C01778=1020.388,138.812,-115.444,167.637,51.113,159.489
C01779=1020.383,138.562,-115.424,167.634,51.119,159.489
C01780=1020.377,138.313,-115.404,167.630,51.126,159.490
C01781=1020.372,138.063,-115.384,167.627,51.133,159.491
C01782=1020.366,137.814,-115.364,167.624,51.140,159.492
C01783=1020.361,137.565,-115.344,167.621,51.147,159.493
C01784=1020.356,137.316,-115.324,167.618,51.154,159.493
C01785=1020.350,137.067,-115.305,167.614,51.160,159.494
C01786=1020.345,136.818,-115.285,167.611,51.167,159.495
C01787=1020.339,136.568,-115.265,167.609,51.174,159.496
C01788=1020.334,136.319,-115.245,167.605,51.181,159.497
C01789=1020.329,136.070,-115.226,167.602,51.188,159.497
C01790=1020.324,135.821,-115.205,167.599,51.195,159.498
C01791=1020.318,135.572,-115.186,167.596,51.201,159.499
C01792=1020.313,135.323,-115.165,167.593,51.208,159.500
C01793=1020.308,135.074,-115.147,167.590,51.215,159.501
C01794=1020.303,134.824,-115.127,167.586,51.222,159.501
C01795=1020.297,134.575,-115.107,167.583,51.229,159.502
C01796=1020.292,134.326,-115.087,167.581,51.236,159.503
C01797=1020.287,134.078,-115.067,167.578,51.243,159.504
C01798=1020.282,133.828,-115.048,167.574,51.250,159.505
C01799=1020.276,133.578,-115.028,167.571,51.257,159.505
C01800=1020.270,133.330,-115.008,167.569,51.263,159.506
C01801=1020.266,133.081,-114.989,167.565,51.270,159.507
C01802=1020.260,132.831,-114.970,167.562,51.277,159.508
C01803=1020.255,132.582,-114.949,167.559,51.284,159.509
C01804=1020.249,132.333,-114.930,167.556,51.290,159.510
C01805=1020.245,132.084,-114.910,167.553,51.297,159.510
C01806=1020.239,131.835,-114.890,167.550,51.304,159.511
C01807=1020.234,131.585,-114.871,167.546,51.311,159.512
C01808=1020.229,131.336,-114.852,167.544,51.318,159.513
C01809=1020.223,131.087,-114.832,167.541,51.325,159.514
C01810=1020.218,130.838,-114.812,167.537,51.331,159.514
C01811=1020.212,130.588,-114.793,167.534,51.338,159.515
C01812=1020.208,130.339,-114.773,167.532,51.345,159.516
C01813=1020.202,130.090,-114.754,167.528,51.352,159.517
C01814=1020.197,129.841,-114.733,167.525,51.359,159.518
C01815=1020.191,129.591,-114.714,167.522,51.366,159.518
C01816=1020.186,129.343,-114.695,167.520,51.373,159.519
C01817=1020.180,129.093,-114.676,167.516,51.380,159.520
C01818=1020.175,128.844,-114.657,167.513,51.387,159.521
C01819=1020.169,128.595,-114.638,167.510,51.394,159.522
C01820=1020.164,128.346,-114.619,167.506,51.401,159.522
C01821=1020.158,128.096,-114.599,167.504,51.407,159.523
C01822=1020.153,127.847,-114.581,167.501,51.415,159.524
C01823=1020.148,127.598,-114.561,167.498,51.422,159.525
C01824=1020.142,127.348,-114.541,167.495,51.429,159.526
C01825=1020.137,127.099,-114.523,167.491,51.436,159.527
C01826=1020.132,126.850,-114.503,167.489,51.442,159.528
C01827=1020.126,126.601,-114.484,167.486,51.450,159.529
C01828=1020.121,126.352,-114.465,167.483,51.457,159.529
C01829=1020.115,126.102,-114.446,167.479,51.464,159.530
C01830=1020.109,125.853,-114.427,167.477,51.470,159.531
C01831=1020.104,125.604,-114.408,167.474,51.477,159.532
C01832=1020.099,125.355,-114.389,167.470,51.484,159.533
C01833=1020.094,125.106,-114.370,167.467,51.491,159.533
C01834=1020.089,124.856,-114.350,167.465,51.498,159.534
C01835=1020.083,124.607,-114.331,167.462,51.505,159.535
C01836=1020.078,124.358,-114.312,167.459,51.512,159.536
C01837=1020.072,124.109,-114.293,167.455,51.519,159.537
C01838=1020.067,123.860,-114.274,167.453,51.526,159.538
C01839=1020.061,123.577,-114.252,167.449,51.534,159.538
C01840=1020.054,123.294,-114.230,167.446,51.541,159.539
C01841=1020.048,123.011,-114.208,167.442,51.549,159.540
C01842=1020.042,122.729,-114.187,167.439,51.557,159.541
C01843=1020.037,122.480,-114.168,167.436,51.564,159.542
C01844=1020.032,122.230,-114.148,167.433,51.571,159.543
C01845=1020.027,121.982,-114.129,167.430,51.578,159.544
C01846=1020.021,121.732,-114.110,167.428,51.585,159.545
C01847=1020.016,121.484,-114.091,167.424,51.592,159.545
C01848=1020.010,121.234,-114.072,167.421,51.599,159.546
C01849=1020.005,120.985,-114.054,167.419,51.606,159.547
C01850=1020.000,120.735,-114.035,167.416,51.612,159.548
C01851=1019.994,120.486,-114.015,167.412,51.619,159.549
C01852=1019.989,120.237,-113.997,167.410,51.626,159.550
C01853=1019.983,119.988,-113.977,167.407,51.633,159.550
C01854=1019.978,119.739,-113.958,167.403,51.640,159.551
C01855=1019.972,119.490,-113.939,167.401,51.647,159.552
C01856=1019.968,119.240,-113.920,167.398,51.654,159.553
C01857=1019.963,118.990,-113.901,167.395,51.660,159.554
C01858=1019.958,118.742,-113.882,167.392,51.667,159.554
C01859=1019.952,118.492,-113.863,167.389,51.675,159.555
C01860=1019.947,118.244,-113.844,167.386,51.682,159.556
C01861=1019.941,117.993,-113.826,167.384,51.688,159.557
C01862=1019.936,117.745,-113.807,167.381,51.695,159.558
C01863=1019.931,117.495,-113.788,167.377,51.702,159.559
C01864=1019.926,117.247,-113.769,167.375,51.709,159.560
C01865=1019.920,116.997,-113.749,167.372,51.716,159.560
C01866=1019.915,116.748,-113.731,167.369,51.723,159.561
C01867=1019.909,116.498,-113.712,167.366,51.729,159.562
C01868=1019.904,116.250,-113.693,167.363,51.736,159.563
C01869=1019.899,116.001,-113.674,167.361,51.743,159.564
C01870=1019.894,115.751,-113.656,167.358,51.750,159.564
C01871=1019.890,115.502,-113.636,167.354,51.757,159.565
C01872=1019.884,115.252,-113.617,167.352,51.764,159.566
C01873=1019.879,115.004,-113.598,167.349,51.771,159.567
C01874=1019.873,114.754,-113.580,167.345,51.778,159.568
C01875=1019.868,114.505,-113.561,167.343,51.784,159.568
C01876=1019.863,114.255,-113.541,167.340,51.791,159.569
C01877=1019.858,114.006,-113.523,167.338,51.798,159.570
C01878=1019.853,113.757,-113.504,167.334,51.804,159.571
C01879=1019.847,113.508,-113.485,167.332,51.811,159.572
C01880=1019.842,113.259,-113.467,167.329,51.818,159.572
C01881=1019.837,113.009,-113.448,167.325,51.825,159.573
C01882=1019.832,112.760,-113.429,167.323,51.831,159.574
C01883=1019.827,112.511,-113.411,167.320,51.838,159.575
C01884=1019.821,112.262,-113.391,167.318,51.845,159.576
C01885=1019.816,112.012,-113.373,167.314,51.852,159.576
C01886=1019.811,111.763,-113.354,167.311,51.859,159.577
C01887=1019.806,111.513,-113.336,167.309,51.866,159.578
C01888=1019.799,111.264,-113.317,167.306,51.873,159.579
C01889=1019.795,111.015,-113.299,167.303,51.880,159.580
C01890=1019.790,110.766,-113.280,167.301,51.887,159.581
C01891=1019.784,110.516,-113.262,167.297,51.894,159.582
C01892=1019.778,110.268,-113.243,167.294,51.901,159.582
C01893=1019.774,110.018,-113.225,167.292,51.908,159.583
C01894=1019.768,109.769,-113.206,167.289,51.915,159.584
C01895=1019.763,109.520,-113.188,167.286,51.921,159.585
C01896=1019.757,109.271,-113.169,167.283,51.928,159.586
C01897=1019.752,109.021,-113.151,167.280,51.935,159.586
C01898=1019.747,108.772,-113.133,167.277,51.943,159.587
C01899=1019.741,108.523,-113.114,167.275,51.950,159.588
C01900=1019.736,108.273,-113.096,167.272,51.957,159.589
C01901=1019.730,108.024,-113.078,167.268,51.964,159.590
C01902=1019.725,107.775,-113.059,167.266,51.970,159.591
C01903=1019.719,107.492,-113.039,167.262,51.978,159.592
C01904=1019.712,107.209,-113.018,167.260,51.986,159.593
C01905=1019.706,106.927,-112.997,167.257,51.994,159.594
C01906=1019.700,106.644,-112.977,167.253,52.002,159.594
C01907=1019.695,106.395,-112.959,167.250,52.009,159.595
C01908=1019.689,106.146,-112.940,167.248,52.016,159.596
C01909=1019.684,105.896,-112.922,167.245,52.023,159.597
C01910=1019.679,105.647,-112.904,167.242,52.030,159.598
C01911=1019.674,105.398,-112.886,167.239,52.037,159.599
C01912=1019.668,105.148,-112.867,167.236,52.044,159.599
C01913=1019.663,104.899,-112.849,167.234,52.050,159.600
C01914=1019.658,104.650,-112.831,167.231,52.057,159.601
C01915=1019.652,104.400,-112.813,167.227,52.064,159.602
C01916=1019.647,104.151,-112.794,167.225,52.071,159.603
C01917=1019.641,103.902,-112.777,167.222,52.078,159.604
C01918=1019.636,103.652,-112.758,167.220,52.085,159.604
C01919=1019.631,103.403,-112.740,167.217,52.093,159.605
C01920=1019.625,103.155,-112.722,167.214,52.100,159.606
C01921=1019.620,102.905,-112.704,167.211,52.106,159.607
C01922=1019.614,102.655,-112.686,167.208,52.113,159.608
C01923=1019.609,102.406,-112.667,167.206,52.120,159.609
C01924=1019.604,102.157,-112.650,167.203,52.127,159.610
C01925=1019.599,101.908,-112.631,167.200,52.134,159.610
C01926=1019.593,101.658,-112.612,167.197,52.141,159.611
C01927=1019.588,101.409,-112.595,167.194,52.148,159.612
C01928=1019.583,101.160,-112.577,167.192,52.154,159.613
C01929=1019.578,100.911,-112.559,167.189,52.161,159.614
C01930=1019.572,100.661,-112.541,167.187,52.168,159.615
C01931=1019.566,100.412,-112.522,167.183,52.175,159.615
C01932=1019.562,100.163,-112.504,167.180,52.182,159.616
C01933=1019.557,99.914,-112.486,167.178,52.189,159.617
C01934=1019.551,99.664,-112.468,167.175,52.196,159.618
C01935=1019.546,99.415,-112.450,167.173,52.203,159.619
C01936=1019.540,99.166,-112.432,167.170,52.210,159.619
C01937=1019.536,98.916,-112.414,167.166,52.217,159.620
C01938=1019.529,98.666,-112.396,167.164,52.223,159.621
C01939=1019.524,98.417,-112.379,167.161,52.230,159.622
C01940=1019.518,98.168,-112.361,167.159,52.237,159.623
C01941=1019.514,97.919,-112.343,167.156,52.245,159.624
C01942=1019.508,97.670,-112.325,167.153,52.252,159.625
C01943=1019.502,97.420,-112.307,167.151,52.259,159.625
C01944=1019.496,97.171,-112.290,167.147,52.266,159.626
C01945=1019.492,96.922,-112.272,167.144,52.273,159.627
C01946=1019.486,96.673,-112.254,167.142,52.279,159.628
C01947=1019.481,96.424,-112.237,167.139,52.286,159.629
C01948=1019.476,96.173,-112.219,167.136,52.293,159.629
C01949=1019.470,95.924,-112.201,167.134,52.301,159.630
C01950=1019.465,95.675,-112.184,167.131,52.308,159.631
C01951=1019.459,95.426,-112.166,167.129,52.315,159.632
C01952=1019.454,95.177,-112.148,167.126,52.322,159.633
C01953=1019.448,94.927,-112.130,167.122,52.329,159.634
C01954=1019.443,94.678,-112.112,167.120,52.335,159.635
C01955=1019.437,94.429,-112.095,167.117,52.343,159.635
C01956=1019.432,94.179,-112.077,167.115,52.349,159.636
C01957=1019.427,93.930,-112.060,167.112,52.356,159.637
C01958=1019.422,93.681,-112.042,167.108,52.363,159.638
C01959=1019.417,93.431,-112.024,167.106,52.370,159.639
C01960=1019.411,93.182,-112.006,167.103,52.377,159.639
C01961=1019.405,92.933,-111.989,167.101,52.384,159.640
C01962=1019.400,92.684,-111.971,167.098,52.391,159.641
C01963=1019.395,92.434,-111.953,167.096,52.398,159.642
C01964=1019.390,92.185,-111.936,167.093,52.405,159.643
C01965=1019.384,91.936,-111.918,167.090,52.412,159.644
C01966=1019.379,91.687,-111.901,167.088,52.419,159.645
C01967=1019.373,91.404,-111.881,167.084,52.426,159.645
C01968=1019.367,91.121,-111.860,167.081,52.434,159.646
C01969=1019.361,90.839,-111.841,167.078,52.442,159.647
C01970=1019.354,90.555,-111.821,167.075,52.450,159.648
C01971=1019.349,90.306,-111.803,167.072,52.457,159.649
C01972=1019.343,90.057,-111.786,167.070,52.464,159.650
C01973=1019.339,89.808,-111.767,167.067,52.471,159.651
C01974=1019.333,89.558,-111.751,167.064,52.478,159.652
C01975=1019.328,89.309,-111.733,167.062,52.485,159.652
C01976=1019.323,89.060,-111.715,167.058,52.492,159.653
C01977=1019.317,88.811,-111.699,167.056,52.498,159.654
C01978=1019.312,88.561,-111.681,167.054,52.506,159.655
C01979=1019.306,88.312,-111.663,167.050,52.513,159.656
C01980=1019.301,88.063,-111.647,167.048,52.520,159.657
C01981=1019.295,87.813,-111.629,167.045,52.527,159.658
C01982=1019.290,87.563,-111.612,167.043,52.534,159.658
C01983=1019.284,87.314,-111.594,167.040,52.541,159.659
C01984=1019.279,87.065,-111.577,167.037,52.548,159.660
C01985=1019.273,86.816,-111.560,167.035,52.555,159.661
C01986=1019.268,86.567,-111.542,167.032,52.563,159.662
C01987=1019.263,86.317,-111.525,167.029,52.570,159.663
C01988=1019.257,86.068,-111.508,167.027,52.576,159.664
C01989=1019.252,85.818,-111.491,167.023,52.583,159.664
C01990=1019.246,85.569,-111.473,167.021,52.590,159.665
C01991=1019.241,85.320,-111.457,167.018,52.597,159.666
C01992=1019.236,85.070,-111.439,167.015,52.604,159.667
C01993=1019.230,84.821,-111.422,167.013,52.611,159.668
C01994=1019.225,84.572,-111.405,167.010,52.618,159.668
C01995=1019.220,84.322,-111.388,167.008,52.625,159.669
C01996=1019.214,84.073,-111.370,167.005,52.633,159.670
C01997=1019.208,83.824,-111.354,167.002,52.640,159.671
C01998=1019.203,83.575,-111.336,167.000,52.647,159.672
C01999=1019.197,83.325,-111.320,166.997,52.654,159.673
C02000=1019.192,83.076,-111.302,166.995,52.661,159.674
C02001=1019.187,82.826,-111.285,166.991,52.668,159.674
C02002=1019.181,82.577,-111.268,166.989,52.674,159.675
C02003=1019.176,82.328,-111.251,166.986,52.681,159.676
C02004=1019.171,82.078,-111.234,166.983,52.689,159.677
C02005=1019.165,81.829,-111.216,166.981,52.695,159.678
C02006=1019.160,81.579,-111.199,166.978,52.702,159.679
C02007=1019.155,81.330,-111.182,166.976,52.709,159.679
C02008=1019.149,81.081,-111.165,166.973,52.716,159.680
C02009=1019.144,80.832,-111.147,166.971,52.723,159.681
C02010=1019.139,80.582,-111.131,166.967,52.730,159.682
C02011=1019.133,80.332,-111.114,166.964,52.737,159.683
C02012=1019.128,80.083,-111.096,166.962,52.744,159.684
C02013=1019.123,79.834,-111.079,166.959,52.751,159.684
C02014=1019.116,79.585,-111.062,166.957,52.758,159.685
C02015=1019.111,79.335,-111.045,166.954,52.765,159.686
C02016=1019.106,79.085,-111.029,166.952,52.772,159.687
C02017=1019.100,78.836,-111.011,166.949,52.779,159.688
C02018=1019.095,78.587,-110.994,166.947,52.786,159.689
C02019=1019.091,78.338,-110.978,166.943,52.793,159.689
C02020=1019.085,78.089,-110.960,166.941,52.800,159.690
C02021=1019.080,77.839,-110.943,166.938,52.807,159.691
C02022=1019.075,77.589,-110.926,166.936,52.813,159.692
C02023=1019.069,77.340,-110.909,166.933,52.821,159.693
C02024=1019.064,77.091,-110.892,166.931,52.827,159.694
C02025=1019.058,76.841,-110.876,166.928,52.835,159.694
C02026=1019.052,76.592,-110.858,166.925,52.842,159.695
C02027=1019.047,76.343,-110.841,166.923,52.848,159.696
C02028=1019.042,76.093,-110.825,166.920,52.856,159.697
C02029=1019.036,75.844,-110.808,166.918,52.862,159.698
C02030=1019.031,75.594,-110.791,166.914,52.869,159.699
C02031=1019.025,75.313,-110.772,166.912,52.877,159.700
C02032=1019.019,75.030,-110.753,166.908,52.886,159.700
C02033=1019.013,74.747,-110.734,166.906,52.893,159.701
C02034=1019.007,74.465,-110.716,166.903,52.901,159.702
C02035=1019.001,74.215,-110.699,166.900,52.908,159.703
C02036=1018.996,73.966,-110.682,166.897,52.916,159.704
C02037=1018.991,73.716,-110.666,166.895,52.922,159.705
C02038=1018.984,73.467,-110.649,166.892,52.929,159.706
C02039=1018.979,73.218,-110.632,166.889,52.936,159.706
C02040=1018.974,72.968,-110.615,166.886,52.943,159.707
C02041=1018.969,72.719,-110.599,166.884,52.950,159.708
C02042=1018.963,72.470,-110.582,166.881,52.957,159.709
C02043=1018.957,72.220,-110.566,166.878,52.964,159.710
C02044=1018.952,71.971,-110.549,166.876,52.971,159.711
C02045=1018.947,71.721,-110.532,166.873,52.978,159.711
C02046=1018.941,71.472,-110.516,166.871,52.985,159.712
C02047=1018.936,71.223,-110.499,166.868,52.992,159.713
C02048=1018.931,70.973,-110.483,166.866,52.999,159.714
C02049=1018.925,70.724,-110.466,166.863,53.006,159.715
C02050=1018.920,70.474,-110.449,166.860,53.013,159.716
C02051=1018.914,70.225,-110.433,166.858,53.020,159.716
C02052=1018.909,69.975,-110.416,166.855,53.027,159.717
C02053=1018.904,69.726,-110.400,166.853,53.034,159.718
C02054=1018.898,69.477,-110.384,166.849,53.041,159.719
C02055=1018.893,69.227,-110.367,166.847,53.048,159.720
C02056=1018.887,68.978,-110.351,166.844,53.055,159.721
C02057=1018.882,68.728,-110.334,166.842,53.062,159.721
C02058=1018.877,68.479,-110.317,166.839,53.069,159.722
C02059=1018.871,68.230,-110.301,166.836,53.076,159.723
C02060=1018.866,67.980,-110.284,166.834,53.083,159.724
C02061=1018.860,67.731,-110.268,166.831,53.090,159.725
C02062=1018.855,67.481,-110.251,166.829,53.097,159.726
C02063=1018.850,67.232,-110.235,166.826,53.104,159.726
C02064=1018.844,66.983,-110.218,166.823,53.112,159.727
C02065=1018.838,66.733,-110.202,166.821,53.118,159.728
C02066=1018.833,66.484,-110.186,166.818,53.126,159.729
C02067=1018.828,66.234,-110.170,166.816,53.132,159.730
C02068=1018.822,65.985,-110.154,166.813,53.140,159.730
C02069=1018.817,65.735,-110.137,166.811,53.146,159.731
C02070=1018.811,65.486,-110.121,166.808,53.153,159.732
C02071=1018.806,65.237,-110.104,166.805,53.161,159.733
C02072=1018.801,64.988,-110.088,166.803,53.167,159.734
C02073=1018.795,64.738,-110.072,166.800,53.175,159.735
C02074=1018.790,64.488,-110.055,166.798,53.181,159.736
C02075=1018.784,64.240,-110.040,166.795,53.189,159.736
C02076=1018.779,63.990,-110.023,166.791,53.196,159.737
C02077=1018.773,63.741,-110.006,166.789,53.203,159.738
C02078=1018.768,63.491,-109.991,166.786,53.210,159.739
C02079=1018.763,63.242,-109.974,166.784,53.217,159.740
C02080=1018.757,62.992,-109.958,166.781,53.224,159.740
C02081=1018.752,62.743,-109.941,166.779,53.231,159.741
C02082=1018.746,62.493,-109.926,166.776,53.238,159.742
C02083=1018.741,62.244,-109.910,166.774,53.246,159.743
C02084=1018.735,61.994,-109.894,166.772,53.253,159.744
C02085=1018.729,61.745,-109.878,166.769,53.260,159.745
C02086=1018.724,61.496,-109.862,166.766,53.267,159.746
C02087=1018.718,61.246,-109.847,166.763,53.274,159.746
C02088=1018.712,60.997,-109.830,166.761,53.281,159.747
C02089=1018.707,60.747,-109.815,166.758,53.288,159.748
C02090=1018.701,60.498,-109.799,166.755,53.296,159.749
C02091=1018.696,60.248,-109.783,166.753,53.303,159.750
C02092=1018.690,59.998,-109.767,166.750,53.310,159.751
C02093=1018.685,59.750,-109.751,166.747,53.317,159.752
C02094=1018.679,59.500,-109.735,166.745,53.324,159.752
C02095=1018.673,59.232,-109.718,166.742,53.332,159.753
C02096=1018.667,58.963,-109.701,166.739,53.339,159.754
C02097=1018.661,58.695,-109.684,166.737,53.347,159.755
C02098=1018.655,58.426,-109.667,166.733,53.355,159.756
C02099=1018.649,58.176,-109.651,166.731,53.362,159.757
C02100=1018.644,57.926,-109.635,166.728,53.370,159.758
C02101=1018.638,57.678,-109.619,166.726,53.376,159.759
C02102=1018.633,57.428,-109.604,166.723,53.384,159.759
C02103=1018.627,57.179,-109.588,166.720,53.391,159.760
C02104=1018.622,56.929,-109.572,166.718,53.398,159.761
C02105=1018.617,56.679,-109.556,166.715,53.405,159.762
C02106=1018.612,56.430,-109.540,166.712,53.412,159.763
C02107=1018.606,56.180,-109.525,166.710,53.419,159.764
C02108=1018.600,55.931,-109.509,166.707,53.426,159.764
C02109=1018.595,55.681,-109.493,166.704,53.433,159.765
C02110=1018.589,55.432,-109.477,166.702,53.440,159.766
C02111=1018.584,55.183,-109.462,166.699,53.447,159.767
C02112=1018.578,54.934,-109.446,166.697,53.454,159.768
C02113=1018.572,54.684,-109.430,166.694,53.461,159.769
C02114=1018.567,54.435,-109.414,166.691,53.469,159.769
C02115=1018.561,54.185,-109.399,166.689,53.476,159.770
C02116=1018.556,53.936,-109.384,166.686,53.483,159.771
C02117=1018.551,53.686,-109.367,166.684,53.490,159.772
C02118=1018.545,53.436,-109.351,166.681,53.497,159.773
C02119=1018.540,53.187,-109.335,166.678,53.504,159.773
C02120=1018.534,52.937,-109.320,166.676,53.511,159.774
C02121=1018.529,52.688,-109.305,166.673,53.518,159.775
C02122=1018.523,52.439,-109.288,166.671,53.525,159.776
C02123=1018.518,52.175,-109.272,166.668,53.532,159.777
C02124=1018.511,51.912,-109.255,166.665,53.539,159.778
C02125=1018.506,51.649,-109.239,166.663,53.547,159.779
C02126=1018.500,51.385,-109.222,166.660,53.555,159.779
C02127=1018.495,51.136,-109.206,166.657,53.562,159.780
C02128=1018.489,50.886,-109.191,166.655,53.569,159.781
C02129=1018.484,50.637,-109.176,166.652,53.576,159.782
C02130=1018.478,50.388,-109.159,166.650,53.583,159.783
C02131=1018.473,50.138,-109.144,166.647,53.590,159.784
C02132=1018.468,49.889,-109.129,166.645,53.597,159.784
C02133=1018.462,49.640,-109.113,166.642,53.603,159.785
C02134=1018.457,49.390,-109.097,166.639,53.611,159.786
C02135=1018.452,49.140,-109.082,166.637,53.618,159.787
C02136=1018.447,48.890,-109.066,166.634,53.625,159.787
C02137=1018.441,48.642,-109.050,166.632,53.632,159.788
C02138=1018.436,48.392,-109.035,166.629,53.639,159.789
C02139=1018.431,48.142,-109.019,166.627,53.646,159.790
C02140=1018.425,47.893,-109.003,166.623,53.652,159.791
C02141=1018.420,47.644,-108.988,166.620,53.660,159.791
C02142=1018.414,47.394,-108.972,166.618,53.666,159.792
C02143=1018.409,47.145,-108.957,166.615,53.674,159.793
C02144=1018.403,46.895,-108.941,166.613,53.681,159.794
C02145=1018.398,46.646,-108.926,166.611,53.688,159.795
C02146=1018.392,46.396,-108.910,166.608,53.694,159.795
C02147=1018.387,46.147,-108.895,166.605,53.701,159.796
C02148=1018.381,45.897,-108.879,166.603,53.708,159.797
C02149=1018.376,45.648,-108.864,166.600,53.715,159.798
C02150=1018.371,45.398,-108.848,166.598,53.722,159.799
C02151=1018.366,45.149,-108.833,166.595,53.729,159.799
C02152=1018.361,44.900,-108.816,166.593,53.736,159.800
C02153=1018.355,44.650,-108.801,166.590,53.743,159.801
C02154=1018.350,44.401,-108.786,166.588,53.750,159.802
C02155=1018.345,44.151,-108.770,166.585,53.756,159.803
C02156=1018.340,43.901,-108.755,166.583,53.763,159.803
C02157=1018.335,43.652,-108.740,166.580,53.771,159.804
C02158=1018.329,43.403,-108.724,166.577,53.778,159.805
C02159=1018.323,43.120,-108.706,166.574,53.785,159.806
C02160=1018.317,42.838,-108.689,166.571,53.793,159.807
C02161=1018.311,42.554,-108.671,166.568,53.800,159.808
C02162=1018.305,42.272,-108.653,166.566,53.808,159.809
C02163=1018.300,42.023,-108.638,166.563,53.816,159.809
C02164=1018.293,41.773,-108.623,166.560,53.823,159.810
C02165=1018.288,41.524,-108.608,166.558,53.830,159.811
C02166=1018.283,41.275,-108.593,166.555,53.837,159.812
C02167=1018.278,41.025,-108.577,166.552,53.844,159.813
C02168=1018.272,40.776,-108.563,166.550,53.850,159.813
C02169=1018.266,40.526,-108.547,166.547,53.858,159.814
C02170=1018.261,40.276,-108.532,166.545,53.865,159.815
C02171=1018.256,40.027,-108.518,166.542,53.872,159.816
C02172=1018.250,39.777,-108.503,166.539,53.879,159.817
C02173=1018.245,39.528,-108.488,166.537,53.886,159.817
C02174=1018.240,39.278,-108.472,166.534,53.893,159.818
C02175=1018.234,39.028,-108.457,166.532,53.900,159.819
C02176=1018.228,38.779,-108.442,166.529,53.907,159.820
C02177=1018.223,38.530,-108.427,166.526,53.914,159.820
C02178=1018.218,38.280,-108.412,166.524,53.921,159.821
C02179=1018.213,38.031,-108.396,166.521,53.928,159.822
C02180=1018.206,37.781,-108.381,166.519,53.935,159.823
C02181=1018.201,37.532,-108.366,166.516,53.942,159.824
C02182=1018.196,37.283,-108.351,166.514,53.949,159.825
C02183=1018.191,37.033,-108.336,166.511,53.956,159.825
C02184=1018.185,36.783,-108.322,166.508,53.963,159.826
C02185=1018.180,36.534,-108.307,166.506,53.970,159.827
C02186=1018.174,36.284,-108.291,166.503,53.977,159.828
C02187=1018.169,36.035,-108.276,166.501,53.984,159.828
C02188=1018.164,35.785,-108.262,166.498,53.991,159.829
C02189=1018.158,35.535,-108.247,166.495,53.998,159.830
C02190=1018.152,35.286,-108.232,166.493,54.005,159.831
C02191=1018.147,35.037,-108.217,166.490,54.013,159.832
C02192=1018.141,34.787,-108.202,166.487,54.020,159.832
C02193=1018.136,34.538,-108.188,166.486,54.027,159.833
C02194=1018.131,34.288,-108.173,166.483,54.034,159.834
C02195=1018.125,34.039,-108.158,166.480,54.041,159.835
C02196=1018.119,33.789,-108.143,166.478,54.048,159.836
C02197=1018.114,33.540,-108.129,166.474,54.055,159.836
C02198=1018.109,33.291,-108.114,166.472,54.062,159.837
C02199=1018.103,33.040,-108.099,166.470,54.069,159.838
C02200=1018.097,32.791,-108.084,166.467,54.076,159.839
C02201=1018.092,32.542,-108.070,166.464,54.084,159.840
C02202=1018.087,32.292,-108.055,166.462,54.091,159.841
C02203=1018.081,32.043,-108.040,166.459,54.098,159.841
C02204=1018.076,31.793,-108.025,166.456,54.105,159.842
C02205=1018.070,31.544,-108.011,166.454,54.111,159.843
C02206=1018.065,31.295,-107.996,166.451,54.119,159.844
C02207=1018.059,31.045,-107.981,166.449,54.126,159.845
C02208=1018.054,30.795,-107.967,166.446,54.133,159.845
C02209=1018.048,30.546,-107.952,166.443,54.140,159.846
C02210=1018.043,30.296,-107.937,166.441,54.147,159.847
C02211=1018.038,30.047,-107.923,166.438,54.154,159.848
C02212=1018.032,29.797,-107.907,166.435,54.161,159.848
C02213=1018.026,29.548,-107.893,166.433,54.168,159.849
C02214=1018.021,29.298,-107.878,166.430,54.175,159.850
C02215=1018.016,29.049,-107.864,166.428,54.182,159.851
C02216=1018.010,28.799,-107.849,166.425,54.189,159.852
C02217=1018.005,28.550,-107.834,166.422,54.196,159.852
C02218=1018.000,28.300,-107.820,166.420,54.203,159.853
C02219=1017.994,28.051,-107.805,166.417,54.210,159.854
C02220=1017.989,27.801,-107.791,166.415,54.217,159.855
C02221=1017.983,27.551,-107.776,166.412,54.224,159.855
C02222=1017.978,27.302,-107.761,166.409,54.231,159.856
C02223=1017.972,27.019,-107.745,166.407,54.239,159.857
C02224=1017.966,26.736,-107.728,166.403,54.247,159.858
C02225=1017.959,26.454,-107.712,166.401,54.255,159.859
C02226=1017.953,26.171,-107.696,166.398,54.263,159.860
C02227=1017.948,25.922,-107.681,166.395,54.270,159.860
C02228=1017.942,25.672,-107.667,166.392,54.277,159.861
C02229=1017.937,25.422,-107.653,166.390,54.284,159.862
C02230=1017.932,25.173,-107.638,166.387,54.292,159.863
C02231=1017.926,24.924,-107.624,166.384,54.299,159.864
C02232=1017.920,24.673,-107.610,166.383,54.306,159.865
C02233=1017.914,24.424,-107.595,166.379,54.312,159.865
C02234=1017.910,24.174,-107.581,166.376,54.320,159.866
C02235=1017.904,23.926,-107.566,166.375,54.327,159.867
C02236=1017.898,23.676,-107.553,166.372,54.334,159.868
C02237=1017.893,23.426,-107.539,166.369,54.341,159.868
C02238=1017.888,23.177,-107.523,166.366,54.348,159.869
C02239=1017.882,22.928,-107.510,166.364,54.355,159.870
C02240=1017.876,22.677,-107.495,166.361,54.362,159.871
C02241=1017.870,22.428,-107.481,166.359,54.369,159.872
C02242=1017.866,22.178,-107.466,166.356,54.377,159.872
C02243=1017.860,21.929,-107.452,166.353,54.383,159.873
C02244=1017.855,21.679,-107.439,166.351,54.390,159.874
C02245=1017.849,21.430,-107.424,166.348,54.398,159.875
C02246=1017.844,21.180,-107.410,166.345,54.405,159.875
C02247=1017.839,20.931,-107.396,166.343,54.411,159.876
C02248=1017.833,20.682,-107.381,166.340,54.419,159.877
C02249=1017.827,20.432,-107.367,166.337,54.426,159.878
C02250=1017.823,20.182,-107.353,166.335,54.433,159.879
C02251=1017.817,19.932,-107.339,166.332,54.440,159.879
C02252=1017.811,19.683,-107.324,166.329,54.447,159.880
C02253=1017.805,19.434,-107.310,166.327,54.454,159.881
C02254=1017.801,19.184,-107.296,166.324,54.461,159.881
C02255=1017.795,18.934,-107.282,166.322,54.467,159.882
C02256=1017.790,18.685,-107.268,166.319,54.475,159.883
C02257=1017.784,18.436,-107.253,166.317,54.482,159.884
C02258=1017.778,18.186,-107.240,166.314,54.490,159.885
C02259=1017.773,17.936,-107.226,166.311,54.496,159.885
C02260=1017.768,17.687,-107.212,166.309,54.503,159.886
C02261=1017.762,17.437,-107.198,166.306,54.511,159.887
C02262=1017.757,17.188,-107.184,166.304,54.518,159.888
C02263=1017.751,16.938,-107.170,166.301,54.524,159.888
C02264=1017.746,16.689,-107.155,166.298,54.532,159.889
C02265=1017.741,16.439,-107.141,166.296,54.539,159.890
C02266=1017.735,16.190,-107.127,166.293,54.546,159.891
C02267=1017.730,15.940,-107.113,166.290,54.553,159.891
C02268=1017.724,15.691,-107.100,166.288,54.560,159.892
C02269=1017.719,15.441,-107.086,166.285,54.567,159.893
C02270=1017.713,15.191,-107.072,166.282,54.574,159.894
C02271=1017.708,14.942,-107.058,166.280,54.581,159.895
C02272=1017.702,14.692,-107.044,166.277,54.588,159.895
C02273=1017.697,14.443,-107.030,166.274,54.595,159.896
C02274=1017.691,14.193,-107.016,166.272,54.602,159.897
C02275=1017.686,13.944,-107.003,166.269,54.609,159.898
C02276=1017.680,13.694,-106.989,166.266,54.616,159.898
C02277=1017.676,13.444,-106.974,166.264,54.623,159.899
C02278=1017.670,13.195,-106.960,166.261,54.630,159.900
C02279=1017.664,12.945,-106.947,166.259,54.637,159.901
C02280=1017.658,12.696,-106.933,166.256,54.645,159.901
C02281=1017.653,12.446,-106.919,166.253,54.651,159.902
C02282=1017.647,12.197,-106.905,166.251,54.658,159.903
C02283=1017.642,11.947,-106.892,166.248,54.666,159.904
C02284=1017.636,11.698,-106.878,166.245,54.673,159.904
C02285=1017.631,11.448,-106.865,166.243,54.680,159.905
C02286=1017.625,11.198,-106.851,166.240,54.688,159.906
C02287=1017.619,10.918,-106.836,166.237,54.695,159.907
C02288=1017.614,10.636,-106.821,166.234,54.703,159.908
C02289=1017.607,10.355,-106.805,166.231,54.712,159.909
C02290=1017.601,10.074,-106.790,166.228,54.719,159.909
C02291=1017.595,9.824,-106.776,166.225,54.727,159.910
C02292=1017.590,9.575,-106.763,166.222,54.734,159.911
C02293=1017.584,9.325,-106.749,166.221,54.741,159.912
C02294=1017.578,9.075,-106.736,166.217,54.748,159.912
C02295=1017.573,8.826,-106.722,166.215,54.755,159.913
C02296=1017.567,8.576,-106.708,166.212,54.763,159.914
C02297=1017.562,8.326,-106.695,166.210,54.770,159.915
C02298=1017.556,8.077,-106.682,166.207,54.776,159.915
C02299=1017.551,7.828,-106.669,166.204,54.784,159.916
C02300=1017.546,7.578,-106.655,166.201,54.791,159.917
C02301=1017.540,7.328,-106.641,166.199,54.797,159.918
C02302=1017.535,7.079,-106.628,166.196,54.805,159.918
C02303=1017.529,6.829,-106.614,166.193,54.812,159.919
C02304=1017.523,6.580,-106.600,166.192,54.819,159.920
C02305=1017.518,6.330,-106.587,166.188,54.826,159.921
C02306=1017.513,6.081,-106.574,166.185,54.833,159.922
C02307=1017.508,5.831,-106.560,166.183,54.841,159.922
C02308=1017.501,5.582,-106.547,166.180,54.847,159.923
C02309=1017.496,5.332,-106.534,166.178,54.854,159.924
C02310=1017.491,5.082,-106.520,166.175,54.862,159.925
C02311=1017.485,4.833,-106.506,166.173,54.868,159.925
C02312=1017.480,4.583,-106.494,166.170,54.876,159.926
C02313=1017.475,4.334,-106.480,166.167,54.883,159.927
C02314=1017.469,4.084,-106.466,166.164,54.890,159.927
C02315=1017.464,3.834,-106.453,166.162,54.897,159.928
C02316=1017.458,3.584,-106.439,166.159,54.903,159.929
C02317=1017.453,3.336,-106.426,166.156,54.911,159.930
C02318=1017.448,3.086,-106.413,166.154,54.918,159.931
C02319=1017.442,2.836,-106.399,166.151,54.925,159.931
C02320=1017.437,2.586,-106.386,166.148,54.932,159.932
C02321=1017.431,2.337,-106.373,166.146,54.938,159.933
C02322=1017.426,2.088,-106.359,166.143,54.946,159.933
C02323=1017.421,1.838,-106.346,166.140,54.953,159.934
C02324=1017.415,1.588,-106.332,166.137,54.960,159.935
C02325=1017.409,1.338,-106.320,166.135,54.967,159.936
C02326=1017.405,1.089,-106.306,166.132,54.974,159.936
C02327=1017.399,0.840,-106.292,166.129,54.981,159.937
C02328=1017.394,0.589,-106.279,166.127,54.987,159.938
C02329=1017.388,0.340,-106.265,166.124,54.995,159.938
C02330=1017.383,0.091,-106.253,166.121,55.002,159.939
C02331=1017.378,-0.159,-106.239,166.119,55.009,159.940
C02332=1017.372,-0.409,-106.226,166.116,55.015,159.940
C02333=1017.367,-0.659,-106.212,166.113,55.023,159.941
C02334=1017.362,-0.908,-106.200,166.111,55.029,159.942
C02335=1017.356,-1.157,-106.186,166.108,55.036,159.943
C02336=1017.351,-1.407,-106.172,166.105,55.043,159.943
C02337=1017.346,-1.656,-106.159,166.103,55.050,159.944
C02338=1017.340,-1.906,-106.146,166.100,55.057,159.945
C02339=1017.335,-2.156,-106.133,166.097,55.064,159.945
C02340=1017.330,-2.405,-106.119,166.095,55.071,159.946
C02341=1017.325,-2.655,-106.106,166.092,55.078,159.947
C02342=1017.318,-2.904,-106.093,166.090,55.084,159.948
C02343=1017.313,-3.154,-106.080,166.087,55.092,159.948
C02344=1017.309,-3.404,-106.067,166.084,55.099,159.949
C02345=1017.303,-3.654,-106.053,166.082,55.105,159.950
C02346=1017.298,-3.904,-106.040,166.079,55.112,159.950
C02347=1017.292,-4.152,-106.027,166.076,55.119,159.951
C02348=1017.287,-4.402,-106.014,166.074,55.126,159.952
C02349=1017.281,-4.652,-106.001,166.071,55.133,159.952
C02350=1017.277,-4.901,-105.988,166.068,55.140,159.953
C02351=1017.270,-5.181,-105.974,166.065,55.148,159.954
C02352=1017.264,-5.460,-105.959,166.062,55.156,159.955
C02353=1017.258,-5.739,-105.945,166.059,55.164,159.956
C02354=1017.252,-6.018,-105.930,166.056,55.172,159.956
C02355=1017.246,-6.268,-105.918,166.053,55.179,159.957
C02356=1017.241,-6.517,-105.905,166.051,55.186,159.958
C02357=1017.236,-6.768,-105.892,166.049,55.194,159.959
C02358=1017.230,-7.017,-105.880,166.045,55.200,159.959
C02359=1017.224,-7.266,-105.867,166.043,55.208,159.960
C02360=1017.219,-7.516,-105.854,166.039,55.215,159.960
C02361=1017.214,-7.765,-105.841,166.038,55.222,159.961
C02362=1017.208,-8.016,-105.828,166.035,55.229,159.962
C02363=1017.203,-8.265,-105.816,166.032,55.236,159.963
C02364=1017.197,-8.515,-105.804,166.029,55.243,159.964
C02365=1017.192,-8.764,-105.790,166.027,55.250,159.964
C02366=1017.186,-9.013,-105.777,166.024,55.257,159.965
C02367=1017.181,-9.264,-105.764,166.021,55.264,159.966
C02368=1017.176,-9.513,-105.752,166.018,55.271,159.966
C02369=1017.170,-9.763,-105.740,166.016,55.278,159.967
C02370=1017.165,-10.013,-105.726,166.013,55.285,159.968
C02371=1017.160,-10.262,-105.714,166.010,55.292,159.968
C02372=1017.154,-10.512,-105.700,166.007,55.299,159.969
C02373=1017.149,-10.761,-105.688,166.005,55.306,159.970
C02374=1017.143,-11.011,-105.676,166.002,55.313,159.971
C02375=1017.138,-11.260,-105.663,165.999,55.320,159.971
C02376=1017.132,-11.510,-105.650,165.996,55.327,159.972
C02377=1017.127,-11.759,-105.638,165.994,55.334,159.973
C02378=1017.122,-12.009,-105.625,165.991,55.341,159.973
C02379=1017.116,-12.259,-105.612,165.988,55.348,159.974
C02380=1017.111,-12.509,-105.600,165.986,55.356,159.975
C02381=1017.106,-12.759,-105.587,165.983,55.362,159.975
C02382=1017.100,-13.008,-105.575,165.981,55.369,159.976
C02383=1017.095,-13.258,-105.562,165.977,55.376,159.977
C02384=1017.090,-13.507,-105.550,165.976,55.383,159.978
C02385=1017.084,-13.757,-105.537,165.973,55.390,159.978
C02386=1017.079,-14.007,-105.524,165.969,55.397,159.979
C02387=1017.073,-14.256,-105.511,165.967,55.404,159.979
C02388=1017.069,-14.505,-105.498,165.964,55.411,159.980
C02389=1017.063,-14.755,-105.486,165.962,55.418,159.981
C02390=1017.057,-15.004,-105.473,165.959,55.425,159.981
C02391=1017.053,-15.254,-105.461,165.956,55.431,159.982
C02392=1017.047,-15.504,-105.448,165.954,55.439,159.983
C02393=1017.042,-15.754,-105.437,165.950,55.445,159.983
C02394=1017.037,-16.004,-105.423,165.947,55.452,159.984
C02395=1017.031,-16.253,-105.411,165.946,55.459,159.985
C02396=1017.025,-16.503,-105.399,165.942,55.466,159.985
C02397=1017.020,-16.752,-105.387,165.940,55.474,159.986
C02398=1017.014,-17.002,-105.374,165.937,55.481,159.987
C02399=1017.009,-17.251,-105.362,165.934,55.488,159.988
C02400=1017.004,-17.501,-105.350,165.932,55.495,159.988
C02401=1016.999,-17.751,-105.337,165.929,55.502,159.989
C02402=1016.993,-18.000,-105.325,165.926,55.509,159.990
C02403=1016.988,-18.250,-105.312,165.923,55.516,159.990
C02404=1016.982,-18.499,-105.300,165.920,55.523,159.991
C02405=1016.977,-18.750,-105.288,165.918,55.530,159.992
C02406=1016.971,-18.999,-105.276,165.916,55.537,159.993
C02407=1016.966,-19.248,-105.264,165.912,55.544,159.993
C02408=1016.960,-19.498,-105.251,165.910,55.552,159.994
C02409=1016.955,-19.748,-105.240,165.906,55.558,159.994
C02410=1016.949,-19.998,-105.227,165.904,55.565,159.995
C02411=1016.944,-20.247,-105.215,165.902,55.572,159.996
C02412=1016.940,-20.497,-105.203,165.898,55.579,159.996
C02413=1016.934,-20.747,-105.191,165.896,55.587,159.997
C02414=1016.928,-20.996,-105.178,165.893,55.593,159.998
C02415=1016.922,-21.274,-105.165,165.890,55.601,159.998
C02416=1016.916,-21.551,-105.152,165.887,55.608,159.999
C02417=1016.910,-21.828,-105.139,165.884,55.617,160.000
C02418=1016.905,-22.106,-105.124,165.881,55.625,160.001
C02419=1016.900,-22.356,-105.113,165.878,55.631,160.001
C02420=1016.894,-22.605,-105.100,165.875,55.638,160.002
C02421=1016.888,-22.855,-105.088,165.872,55.646,160.003
C02422=1016.883,-23.104,-105.076,165.870,55.652,160.003
C02423=1016.878,-23.354,-105.064,165.868,55.660,160.004
C02424=1016.872,-23.603,-105.052,165.864,55.666,160.005
C02425=1016.867,-23.853,-105.040,165.861,55.673,160.005
C02426=1016.862,-24.102,-105.028,165.860,55.680,160.006
C02427=1016.856,-24.352,-105.015,165.856,55.687,160.007
C02428=1016.851,-24.602,-105.004,165.853,55.694,160.007
C02429=1016.846,-24.851,-104.992,165.850,55.701,160.008
C02430=1016.841,-25.102,-104.979,165.848,55.708,160.009
C02431=1016.835,-25.351,-104.967,165.845,55.715,160.009
C02432=1016.830,-25.600,-104.955,165.842,55.721,160.010
C02433=1016.825,-25.850,-104.944,165.839,55.729,160.011
C02434=1016.819,-26.100,-104.931,165.837,55.735,160.011
C02435=1016.814,-26.350,-104.920,165.834,55.742,160.012
C02436=1016.809,-26.599,-104.907,165.831,55.750,160.013
C02437=1016.804,-26.849,-104.896,165.829,55.756,160.013
C02438=1016.798,-27.099,-104.883,165.826,55.763,160.014
C02439=1016.793,-27.349,-104.872,165.823,55.770,160.014
C02440=1016.788,-27.598,-104.860,165.820,55.777,160.015
C02441=1016.782,-27.848,-104.848,165.818,55.784,160.016
C02442=1016.777,-28.098,-104.836,165.815,55.790,160.016
C02443=1016.772,-28.347,-104.824,165.812,55.798,160.017
C02444=1016.767,-28.597,-104.813,165.809,55.805,160.018
C02445=1016.761,-28.846,-104.801,165.807,55.812,160.018
C02446=1016.755,-29.096,-104.789,165.803,55.819,160.019
C02447=1016.750,-29.346,-104.777,165.801,55.826,160.020
C02448=1016.745,-29.595,-104.766,165.799,55.833,160.020
C02449=1016.740,-29.845,-104.754,165.795,55.840,160.021
C02450=1016.733,-30.095,-104.742,165.793,55.847,160.022
C02451=1016.728,-30.345,-104.731,165.790,55.854,160.022
C02452=1016.723,-30.594,-104.719,165.787,55.861,160.023
C02453=1016.718,-30.844,-104.707,165.785,55.868,160.024
C02454=1016.713,-31.093,-104.696,165.782,55.875,160.024
C02455=1016.707,-31.343,-104.685,165.779,55.882,160.025
C02456=1016.701,-31.593,-104.673,165.776,55.889,160.026
C02457=1016.696,-31.843,-104.661,165.773,55.896,160.026
C02458=1016.691,-32.092,-104.649,165.771,55.903,160.027
C02459=1016.686,-32.342,-104.638,165.768,55.910,160.028
C02460=1016.680,-32.592,-104.627,165.765,55.917,160.028
C02461=1016.675,-32.841,-104.615,165.762,55.924,160.029
C02462=1016.670,-33.091,-104.603,165.759,55.931,160.029
C02463=1016.665,-33.341,-104.591,165.757,55.938,160.030
C02464=1016.659,-33.591,-104.580,165.754,55.945,160.031
C02465=1016.653,-33.840,-104.568,165.751,55.951,160.031
C02466=1016.648,-34.090,-104.557,165.748,55.959,160.032
C02467=1016.643,-34.339,-104.545,165.746,55.965,160.033
C02468=1016.638,-34.589,-104.534,165.743,55.972,160.033
C02469=1016.632,-34.838,-104.522,165.740,55.979,160.034
C02470=1016.627,-35.088,-104.511,165.737,55.987,160.034
C02471=1016.622,-35.338,-104.499,165.734,55.993,160.035
C02472=1016.617,-35.588,-104.487,165.732,56.000,160.036
C02473=1016.611,-35.838,-104.477,165.729,56.007,160.036
C02474=1016.606,-36.088,-104.465,165.726,56.014,160.037
C02475=1016.601,-36.337,-104.453,165.723,56.021,160.037
C02476=1016.596,-36.587,-104.441,165.721,56.028,160.038
C02477=1016.591,-36.836,-104.430,165.718,56.034,160.039
C02478=1016.585,-37.086,-104.419,165.715,56.041,160.039
C02479=1016.579,-37.362,-104.406,165.712,56.049,160.040
C02480=1016.573,-37.639,-104.394,165.708,56.057,160.041
C02481=1016.568,-37.915,-104.381,165.706,56.064,160.041
C02482=1016.562,-38.191,-104.368,165.703,56.071,160.042
C02483=1016.557,-38.441,-104.357,165.700,56.079,160.043
C02484=1016.552,-38.690,-104.345,165.697,56.086,160.043
C02485=1016.547,-38.940,-104.334,165.695,56.092,160.044
C02486=1016.541,-39.190,-104.323,165.692,56.099,160.044
C02487=1016.536,-39.440,-104.312,165.689,56.106,160.045
C02488=1016.531,-39.689,-104.300,165.685,56.113,160.045
C02489=1016.525,-39.939,-104.289,165.683,56.120,160.046
C02490=1016.520,-40.189,-104.278,165.681,56.127,160.047
C02491=1016.515,-40.438,-104.267,165.678,56.134,160.047
C02492=1016.510,-40.688,-104.255,165.675,56.140,160.048
C02493=1016.504,-40.937,-104.245,165.672,56.148,160.049
C02494=1016.499,-41.187,-104.233,165.669,56.155,160.049
C02495=1016.493,-41.437,-104.222,165.666,56.162,160.050
C02496=1016.488,-41.687,-104.211,165.663,56.169,160.050
C02497=1016.483,-41.937,-104.201,165.661,56.176,160.051
C02498=1016.478,-42.186,-104.189,165.658,56.183,160.052
C02499=1016.472,-42.436,-104.178,165.655,56.189,160.052
C02500=1016.467,-42.686,-104.167,165.652,56.196,160.053
C02501=1016.461,-42.935,-104.156,165.649,56.204,160.054
C02502=1016.456,-43.185,-104.144,165.647,56.210,160.054
C02503=1016.451,-43.435,-104.134,165.644,56.217,160.055
C02504=1016.446,-43.685,-104.123,165.641,56.224,160.055
C02505=1016.440,-43.934,-104.112,165.638,56.231,160.056
C02506=1016.435,-44.184,-104.100,165.635,56.238,160.057
C02507=1016.429,-44.434,-104.090,165.633,56.245,160.057
C02508=1016.425,-44.684,-104.079,165.630,56.252,160.058
C02509=1016.420,-44.933,-104.068,165.627,56.259,160.058
C02510=1016.415,-45.183,-104.057,165.624,56.266,160.059
C02511=1016.409,-45.432,-104.046,165.621,56.272,160.059
C02512=1016.404,-45.682,-104.034,165.619,56.279,160.060
C02513=1016.398,-45.932,-104.024,165.615,56.286,160.061
C02514=1016.393,-46.182,-104.013,165.613,56.293,160.061
C02515=1016.388,-46.431,-104.002,165.610,56.300,160.062
C02516=1016.383,-46.681,-103.990,165.608,56.307,160.063
C02517=1016.377,-46.931,-103.980,165.605,56.314,160.063
C02518=1016.373,-47.180,-103.969,165.602,56.320,160.064
C02519=1016.367,-47.430,-103.958,165.598,56.327,160.064
C02520=1016.361,-47.679,-103.947,165.595,56.334,160.065
C02521=1016.357,-47.930,-103.937,165.593,56.341,160.065
C02522=1016.351,-48.179,-103.926,165.590,56.348,160.066
C02523=1016.346,-48.429,-103.914,165.587,56.354,160.066
C02524=1016.341,-48.679,-103.905,165.584,56.361,160.067
C02525=1016.336,-48.928,-103.893,165.582,56.368,160.068
///RCONF 1,0,0,1,0,0,0,0,0,0,0,0,0,0,0,0,0,0,0,0,0,0,0,0
C02526=1016.330,-49.178,-103.882,165.579,56.375,160.068
C02527=1016.326,-49.428,-103.871,165.576,56.382,160.069
C02528=1016.320,-49.678,-103.861,165.574,56.388,160.069
C02529=1016.315,-49.927,-103.849,165.571,56.395,160.070
C02530=1016.310,-50.177,-103.839,165.568,56.402,160.070
C02531=1016.305,-50.427,-103.828,165.564,56.409,160.071
C02532=1016.300,-50.677,-103.818,165.562,56.415,160.072
C02533=1016.295,-50.927,-103.806,165.559,56.422,160.072
C02534=1016.289,-51.176,-103.795,165.556,56.429,160.073
C02535=1016.283,-51.426,-103.785,165.553,56.436,160.073
C02536=1016.279,-51.676,-103.775,165.551,56.443,160.074
C02537=1016.273,-51.925,-103.764,165.548,56.450,160.074
C02538=1016.267,-52.175,-103.754,165.545,56.457,160.075
C02539=1016.262,-52.425,-103.743,165.543,56.464,160.076
C02540=1016.258,-52.674,-103.733,165.540,56.471,160.076
C02541=1016.252,-52.925,-103.723,165.537,56.478,160.077
C02542=1016.246,-53.174,-103.712,165.534,56.485,160.077
C02543=1016.241,-53.451,-103.701,165.530,56.493,160.078
C02544=1016.235,-53.728,-103.690,165.528,56.501,160.079
C02545=1016.228,-54.004,-103.678,165.524,56.509,160.079
C02546=1016.223,-54.281,-103.667,165.521,56.516,160.080
C02547=1016.217,-54.530,-103.656,165.518,56.523,160.081
C02548=1016.212,-54.780,-103.646,165.515,56.530,160.081
C02549=1016.207,-55.030,-103.636,165.512,56.537,160.082
C02550=1016.201,-55.279,-103.625,165.509,56.544,160.082
C02551=1016.196,-55.529,-103.615,165.507,56.551,160.083
C02552=1016.191,-55.779,-103.605,165.505,56.558,160.084
C02553=1016.186,-56.029,-103.595,165.501,56.565,160.084
C02554=1016.181,-56.279,-103.584,165.498,56.572,160.085
C02555=1016.175,-56.529,-103.574,165.495,56.579,160.085
C02556=1016.170,-56.778,-103.564,165.492,56.586,160.086
C02557=1016.165,-57.028,-103.554,165.489,56.593,160.086
C02558=1016.159,-57.278,-103.543,165.487,56.599,160.087
C02559=1016.154,-57.527,-103.533,165.484,56.606,160.088
C02560=1016.149,-57.777,-103.523,165.481,56.613,160.088
C02561=1016.144,-58.027,-103.513,165.479,56.621,160.089
C02562=1016.138,-58.276,-103.502,165.475,56.628,160.089
C02563=1016.133,-58.526,-103.492,165.472,56.634,160.090
C02564=1016.128,-58.776,-103.482,165.470,56.641,160.091
C02565=1016.123,-59.026,-103.472,165.467,56.648,160.091
C02566=1016.117,-59.276,-103.462,165.464,56.655,160.092
C02567=1016.112,-59.525,-103.451,165.461,56.662,160.092
C02568=1016.107,-59.775,-103.441,165.458,56.669,160.093
C02569=1016.101,-60.025,-103.431,165.456,56.675,160.093
C02570=1016.097,-60.274,-103.421,165.453,56.682,160.094
C02571=1016.092,-60.525,-103.410,165.450,56.689,160.094
C02572=1016.087,-60.774,-103.401,165.447,56.696,160.095
C02573=1016.081,-61.024,-103.390,165.444,56.703,160.095
C02574=1016.076,-61.273,-103.380,165.442,56.709,160.096
C02575=1016.071,-61.523,-103.370,165.439,56.716,160.097
C02576=1016.066,-61.773,-103.360,165.436,56.723,160.097
C02577=1016.061,-62.023,-103.350,165.432,56.729,160.097
C02578=1016.055,-62.273,-103.340,165.430,56.736,160.098
C02579=1016.050,-62.522,-103.330,165.427,56.743,160.099
C02580=1016.045,-62.772,-103.320,165.424,56.750,160.099
C02581=1016.040,-63.022,-103.310,165.421,56.757,160.100
C02582=1016.034,-63.271,-103.299,165.419,56.763,160.100
C02583=1016.030,-63.521,-103.289,165.416,56.770,160.101
C02584=1016.024,-63.771,-103.279,165.413,56.777,160.101
C02585=1016.019,-64.020,-103.269,165.410,56.784,160.102
C02586=1016.014,-64.270,-103.259,165.408,56.790,160.102
C02587=1016.009,-64.520,-103.249,165.404,56.797,160.103
C02588=1016.004,-64.770,-103.239,165.401,56.804,160.103
C02589=1015.999,-65.019,-103.229,165.398,56.811,160.104
C02590=1015.993,-65.269,-103.219,165.396,56.817,160.104
C02591=1015.989,-65.519,-103.209,165.393,56.824,160.105
C02592=1015.983,-65.769,-103.199,165.390,56.831,160.105
C02593=1015.978,-66.018,-103.189,165.387,56.837,160.106
C02594=1015.973,-66.268,-103.179,165.385,56.844,160.106
C02595=1015.968,-66.518,-103.169,165.382,56.851,160.107
C02596=1015.963,-66.768,-103.159,165.379,56.858,160.107
C02597=1015.958,-67.017,-103.149,165.377,56.864,160.108
C02598=1015.954,-67.267,-103.139,165.373,56.870,160.108
C02599=1015.948,-67.517,-103.129,165.370,56.877,160.109
C02600=1015.943,-67.766,-103.119,165.368,56.884,160.110
C02601=1015.938,-68.016,-103.109,165.365,56.891,160.110
C02602=1015.933,-68.266,-103.099,165.361,56.897,160.110
C02603=1015.928,-68.516,-103.089,165.359,56.903,160.111
C02604=1015.923,-68.765,-103.079,165.356,56.910,160.111
C02605=1015.918,-69.015,-103.070,165.353,56.917,160.112
C02606=1015.913,-69.266,-103.060,165.351,56.923,160.112
C02607=1015.907,-69.543,-103.049,165.347,56.930,160.113
C02608=1015.902,-69.821,-103.038,165.344,56.938,160.114
C02609=1015.896,-70.098,-103.027,165.341,56.945,160.114
C02610=1015.890,-70.376,-103.017,165.337,56.952,160.114
C02611=1015.885,-70.626,-103.006,165.335,56.959,160.115
C02612=1015.880,-70.876,-102.997,165.332,56.966,160.116
C02613=1015.875,-71.125,-102.987,165.330,56.972,160.116
C02614=1015.870,-71.375,-102.977,165.327,56.979,160.116
C02615=1015.865,-71.625,-102.967,165.324,56.986,160.117
C02616=1015.861,-71.875,-102.958,165.321,56.991,160.117
C02617=1015.855,-72.125,-102.948,165.318,56.998,160.118
C02618=1015.850,-72.374,-102.938,165.314,57.005,160.118
C02619=1015.845,-72.624,-102.928,165.312,57.011,160.119
C02620=1015.840,-72.874,-102.918,165.309,57.018,160.119
C02621=1015.836,-73.124,-102.909,165.307,57.024,160.120
C02622=1015.831,-73.373,-102.899,165.304,57.031,160.120
C02623=1015.825,-73.623,-102.889,165.300,57.037,160.120
C02624=1015.820,-73.873,-102.879,165.298,57.044,160.121
C02625=1015.816,-74.122,-102.869,165.295,57.050,160.121
C02626=1015.811,-74.372,-102.860,165.293,57.056,160.122
C02627=1015.806,-74.622,-102.850,165.289,57.063,160.122
C02628=1015.801,-74.872,-102.840,165.286,57.070,160.123
C02629=1015.796,-75.122,-102.831,165.284,57.076,160.124
C02630=1015.791,-75.372,-102.821,165.281,57.083,160.124
C02631=1015.786,-75.622,-102.812,165.278,57.089,160.124
C02632=1015.781,-75.871,-102.803,165.275,57.096,160.125
C02633=1015.776,-76.120,-102.793,165.273,57.103,160.125
C02634=1015.770,-76.371,-102.784,165.270,57.110,160.126
C02635=1015.765,-76.620,-102.774,165.266,57.116,160.126
C02636=1015.761,-76.870,-102.765,165.264,57.123,160.127
C02637=1015.756,-77.120,-102.755,165.261,57.130,160.127
C02638=1015.750,-77.370,-102.746,165.258,57.136,160.128
C02639=1015.745,-77.620,-102.737,165.256,57.142,160.128
C02640=1015.741,-77.870,-102.728,165.253,57.149,160.129
C02641=1015.735,-78.119,-102.718,165.249,57.156,160.129
C02642=1015.731,-78.369,-102.709,165.247,57.162,160.130
C02643=1015.725,-78.619,-102.699,165.244,57.169,160.130
C02644=1015.720,-78.868,-102.691,165.241,57.175,160.130
C02645=1015.715,-79.118,-102.681,165.239,57.182,160.131
C02646=1015.710,-79.368,-102.672,165.236,57.189,160.132
C02647=1015.706,-79.617,-102.662,165.232,57.195,160.132
C02648=1015.700,-79.867,-102.654,165.230,57.202,160.133
C02649=1015.695,-80.118,-102.644,165.227,57.208,160.133
C02650=1015.690,-80.367,-102.634,165.224,57.215,160.133
C02651=1015.685,-80.617,-102.626,165.222,57.221,160.134
C02652=1015.680,-80.866,-102.616,165.218,57.228,160.134
C02653=1015.675,-81.116,-102.608,165.215,57.235,160.135
C02654=1015.670,-81.366,-102.599,165.212,57.242,160.135
C02655=1015.665,-81.616,-102.590,165.210,57.248,160.136
C02656=1015.659,-81.866,-102.580,165.207,57.255,160.136
C02657=1015.655,-82.116,-102.571,165.204,57.261,160.137
C02658=1015.649,-82.365,-102.563,165.201,57.268,160.137
C02659=1015.645,-82.615,-102.554,165.199,57.275,160.138
C02660=1015.639,-82.864,-102.545,165.195,57.281,160.138
C02661=1015.634,-83.114,-102.536,165.192,57.288,160.139
C02662=1015.629,-83.364,-102.527,165.189,57.295,160.139
C02663=1015.624,-83.614,-102.519,165.187,57.302,160.140
C02664=1015.620,-83.864,-102.509,165.184,57.308,160.140
C02665=1015.613,-84.114,-102.500,165.181,57.315,160.141
C02666=1015.608,-84.363,-102.491,165.179,57.322,160.141
C02667=1015.604,-84.613,-102.482,165.175,57.328,160.141
C02668=1015.598,-84.863,-102.474,165.172,57.335,160.142
C02669=1015.594,-85.113,-102.465,165.170,57.341,160.143
C02670=1015.589,-85.363,-102.456,165.167,57.348,160.143
C02671=1015.584,-85.584,-102.449,165.164,57.354,160.143
C02672=1015.580,-85.806,-102.440,165.162,57.359,160.144
C02673=1015.575,-86.028,-102.433,165.159,57.365,160.144
C02674=1015.570,-86.249,-102.425,165.157,57.371,160.145
C02675=1015.567,-86.471,-102.417,165.154,57.377,160.145
C02676=1015.562,-86.692,-102.409,165.152,57.383,160.145
C02677=1015.558,-86.913,-102.402,165.149,57.389,160.146
C02678=1015.553,-87.135,-102.393,165.147,57.394,160.146
C02679=1015.548,-87.385,-102.385,165.143,57.401,160.146
C02680=1015.543,-87.635,-102.375,165.140,57.408,160.147
C02681=1015.538,-87.885,-102.367,165.139,57.414,160.148
C02682=1015.532,-88.134,-102.358,165.135,57.421,160.148
C02683=1015.528,-88.384,-102.349,165.132,57.428,160.148
C02684=1015.523,-88.633,-102.341,165.130,57.433,160.149
C02685=1015.519,-88.883,-102.331,165.127,57.440,160.149
C02686=1015.513,-89.133,-102.323,165.124,57.446,160.150
C02687=1015.508,-89.382,-102.315,165.121,57.453,160.150
C02688=1015.504,-89.632,-102.305,165.118,57.460,160.150
C02689=1015.498,-89.882,-102.297,165.116,57.466,160.151
C02690=1015.494,-90.132,-102.288,165.112,57.472,160.151
C02691=1015.489,-90.382,-102.279,165.109,57.479,160.152
C02692=1015.483,-90.632,-102.271,165.107,57.485,160.152
C02693=1015.479,-90.882,-102.262,165.103,57.492,160.152
C02694=1015.474,-91.131,-102.253,165.101,57.498,160.153
C02695=1015.469,-91.381,-102.244,165.098,57.504,160.153
C02696=1015.464,-91.631,-102.236,165.096,57.511,160.154
C02697=1015.459,-91.881,-102.227,165.092,57.517,160.154
C02698=1015.454,-92.131,-102.218,165.089,57.524,160.155
C02699=1015.449,-92.381,-102.210,165.087,57.530,160.155
C02700=1015.445,-92.630,-102.201,165.083,57.536,160.155
C02701=1015.440,-92.880,-102.193,165.082,57.543,160.156
C02702=1015.434,-93.129,-102.184,165.078,57.549,160.156
C02703=1015.430,-93.380,-102.176,165.076,57.555,160.157
C02704=1015.425,-93.630,-102.167,165.073,57.562,160.157
C02705=1015.420,-93.879,-102.159,165.070,57.568,160.158
C02706=1015.415,-94.129,-102.150,165.067,57.574,160.158
C02707=1015.410,-94.378,-102.141,165.065,57.581,160.159
C02708=1015.406,-94.628,-102.132,165.061,57.587,160.159
C02709=1015.401,-94.878,-102.124,165.059,57.593,160.159
C02710=1015.395,-95.128,-102.115,165.056,57.600,160.160
C02711=1015.390,-95.464,-102.104,165.052,57.608,160.160
C02712=1015.383,-95.801,-102.092,165.048,57.617,160.161
C02713=1015.376,-96.137,-102.081,165.044,57.625,160.161
C02714=1015.369,-96.473,-102.069,165.041,57.633,160.162
C02715=1015.365,-96.724,-102.061,165.037,57.640,160.162
C02716=1015.360,-96.973,-102.053,165.035,57.645,160.162
C02717=1015.355,-97.222,-102.044,165.032,57.652,160.163
C02718=1015.351,-97.472,-102.035,165.030,57.658,160.163
C02719=1015.345,-97.722,-102.027,165.026,57.665,160.164
C02720=1015.341,-97.973,-102.018,165.024,57.671,160.164
C02721=1015.336,-98.222,-102.010,165.021,57.678,160.164
C02722=1015.331,-98.472,-102.002,165.018,57.683,160.165
C02723=1015.326,-98.722,-101.994,165.015,57.690,160.165
C02724=1015.321,-98.972,-101.985,165.013,57.696,160.166
C02725=1015.316,-99.221,-101.977,165.009,57.703,160.166
C02726=1015.311,-99.471,-101.970,165.006,57.710,160.166
C02727=1015.306,-99.721,-101.961,165.004,57.716,160.167
C02728=1015.301,-99.971,-101.953,165.000,57.722,160.167
C02729=1015.297,-100.220,-101.945,164.998,57.728,160.168
C02730=1015.292,-100.471,-101.937,164.995,57.735,160.168
C02731=1015.287,-100.720,-101.928,164.993,57.741,160.168
C02732=1015.282,-100.970,-101.920,164.990,57.748,160.169
C02733=1015.277,-101.220,-101.912,164.987,57.754,160.169
C02734=1015.272,-101.469,-101.904,164.984,57.760,160.170
C02735=1015.267,-101.751,-101.895,164.981,57.767,160.170
C02736=1015.262,-102.033,-101.886,164.978,57.774,160.170
C02737=1015.256,-102.315,-101.877,164.975,57.781,160.171
C02738=1015.250,-102.597,-101.868,164.971,57.788,160.171
C02739=1015.246,-102.846,-101.859,164.968,57.794,160.172
C02740=1015.241,-103.097,-101.852,164.965,57.801,160.172
C02741=1015.236,-103.346,-101.843,164.963,57.807,160.173
C02742=1015.231,-103.596,-101.836,164.960,57.814,160.173
C02743=1015.226,-103.846,-101.827,164.957,57.819,160.173
C02744=1015.221,-104.096,-101.819,164.955,57.825,160.174
C02745=1015.217,-104.345,-101.811,164.952,57.832,160.174
C02746=1015.212,-104.595,-101.804,164.949,57.838,160.175
C02747=1015.207,-104.844,-101.795,164.946,57.845,160.175
C02748=1015.202,-105.095,-101.788,164.943,57.850,160.175
C02749=1015.197,-105.345,-101.780,164.940,57.857,160.175
C02750=1015.192,-105.594,-101.772,164.938,57.863,160.176
C02751=1015.187,-105.844,-101.764,164.934,57.870,160.176
C02752=1015.183,-106.094,-101.755,164.932,57.876,160.177
C02753=1015.178,-106.344,-101.747,164.930,57.882,160.177
C02754=1015.174,-106.594,-101.740,164.926,57.888,160.177
C02755=1015.169,-106.843,-101.732,164.924,57.894,160.178
C02756=1015.164,-107.094,-101.724,164.921,57.901,160.178
C02757=1015.159,-107.343,-101.716,164.918,57.907,160.179
C02758=1015.154,-107.593,-101.708,164.915,57.913,160.179
C02759=1015.149,-107.843,-101.700,164.912,57.919,160.179
C02760=1015.145,-108.093,-101.693,164.910,57.925,160.180
C02761=1015.140,-108.343,-101.684,164.906,57.931,160.180
C02762=1015.135,-108.592,-101.677,164.904,57.937,160.180
C02763=1015.130,-108.842,-101.670,164.901,57.944,160.181
C02764=1015.125,-109.092,-101.662,164.899,57.950,160.181
C02765=1015.120,-109.342,-101.654,164.895,57.956,160.181
C02766=1015.116,-109.591,-101.646,164.893,57.962,160.182
C02767=1015.111,-109.842,-101.639,164.889,57.969,160.182
C02768=1015.106,-110.091,-101.631,164.887,57.975,160.183
C02769=1015.101,-110.342,-101.623,164.885,57.981,160.183
C02770=1015.096,-110.590,-101.616,164.882,57.987,160.183
C02771=1015.091,-110.841,-101.608,164.879,57.993,160.184
C02772=1015.087,-111.090,-101.601,164.876,58.000,160.184
C02773=1015.082,-111.341,-101.593,164.873,58.006,160.184
C02774=1015.077,-111.590,-101.586,164.871,58.011,160.185
C02775=1015.072,-111.841,-101.578,164.867,58.018,160.185
C02776=1015.068,-112.090,-101.570,164.865,58.024,160.185
C02777=1015.063,-112.340,-101.562,164.861,58.030,160.185
C02778=1015.058,-112.589,-101.555,164.860,58.037,160.186
C02779=1015.053,-112.840,-101.547,164.857,58.043,160.187
C02780=1015.048,-113.089,-101.540,164.854,58.049,160.187
C02781=1015.044,-113.339,-101.533,164.851,58.055,160.187
C02782=1015.039,-113.589,-101.525,164.849,58.061,160.188
C02783=1015.035,-113.839,-101.517,164.845,58.067,160.188
C02784=1015.030,-114.089,-101.510,164.843,58.073,160.188
C02785=1015.025,-114.338,-101.502,164.840,58.079,160.189
C02786=1015.020,-114.588,-101.495,164.837,58.085,160.189
C02787=1015.015,-114.838,-101.487,164.835,58.091,160.189
C02788=1015.011,-115.088,-101.480,164.832,58.097,160.190
C02789=1015.006,-115.338,-101.472,164.829,58.103,160.190
C02790=1015.001,-115.588,-101.464,164.826,58.109,160.190
C02791=1014.996,-115.837,-101.458,164.824,58.115,160.191
C02792=1014.992,-116.088,-101.450,164.820,58.121,160.191
C02793=1014.987,-116.337,-101.443,164.818,58.127,160.191
C02794=1014.982,-116.588,-101.435,164.816,58.133,160.192
C02795=1014.977,-116.837,-101.429,164.812,58.140,160.192
C02796=1014.973,-117.087,-101.421,164.810,58.146,160.192
C02797=1014.968,-117.337,-101.413,164.807,58.151,160.193
C02798=1014.964,-117.587,-101.406,164.804,58.158,160.193
C02799=1014.958,-117.869,-101.397,164.800,58.164,160.193
C02800=1014.953,-118.151,-101.390,164.797,58.171,160.193
C02801=1014.947,-118.432,-101.382,164.795,58.178,160.194
C02802=1014.941,-118.714,-101.373,164.791,58.185,160.194
C02803=1014.937,-118.964,-101.366,164.789,58.191,160.195
C02804=1014.933,-119.214,-101.359,164.786,58.197,160.195
C02805=1014.928,-119.463,-101.352,164.783,58.203,160.195
C02806=1014.923,-119.714,-101.344,164.780,58.209,160.196
C02807=1014.918,-119.963,-101.337,164.778,58.215,160.196
C02808=1014.914,-120.213,-101.330,164.776,58.221,160.196
C02809=1014.909,-120.464,-101.323,164.772,58.227,160.197
C02810=1014.904,-120.713,-101.316,164.770,58.233,160.197
C02811=1014.900,-120.963,-101.308,164.767,58.238,160.197
C02812=1014.895,-121.212,-101.301,164.764,58.244,160.197
C02813=1014.890,-121.463,-101.294,164.761,58.250,160.198
C02814=1014.886,-121.713,-101.287,164.758,58.256,160.198
C02815=1014.881,-121.962,-101.280,164.756,58.262,160.198
C02816=1014.876,-122.212,-101.273,164.754,58.268,160.199
C02817=1014.871,-122.462,-101.265,164.750,58.274,160.199
C02818=1014.866,-122.712,-101.259,164.748,58.280,160.199
C02819=1014.862,-122.962,-101.252,164.745,58.286,160.200
C02820=1014.858,-123.211,-101.244,164.742,58.292,160.200
C02821=1014.852,-123.462,-101.238,164.740,58.297,160.200
C02822=1014.848,-123.712,-101.230,164.737,58.304,160.201
C02823=1014.843,-123.961,-101.223,164.734,58.310,160.201
C02824=1014.839,-124.211,-101.216,164.731,58.315,160.201
C02825=1014.835,-124.461,-101.209,164.729,58.321,160.201
C02826=1014.829,-124.711,-101.202,164.726,58.327,160.202
C02827=1014.825,-124.961,-101.195,164.723,58.333,160.202
C02828=1014.820,-125.210,-101.189,164.720,58.339,160.202
C02829=1014.815,-125.460,-101.181,164.717,58.344,160.203
C02830=1014.811,-125.710,-101.175,164.715,58.350,160.203
C02831=1014.806,-125.960,-101.168,164.713,58.356,160.203
C02832=1014.801,-126.210,-101.161,164.709,58.362,160.204
C02833=1014.796,-126.460,-101.154,164.707,58.368,160.204
C02834=1014.792,-126.710,-101.148,164.704,58.374,160.204
C02835=1014.787,-126.959,-101.140,164.701,58.380,160.204
C02836=1014.782,-127.209,-101.134,164.699,58.385,160.205
C02837=1014.778,-127.459,-101.127,164.696,58.392,160.205
C02838=1014.774,-127.709,-101.120,164.693,58.398,160.205
C02839=1014.769,-127.959,-101.113,164.690,58.403,160.206
C02840=1014.764,-128.208,-101.107,164.688,58.409,160.206
C02841=1014.760,-128.458,-101.099,164.685,58.414,160.206
C02842=1014.756,-128.708,-101.091,164.683,58.419,160.206
C02843=1014.752,-128.957,-101.083,164.679,58.423,160.206
C02844=1014.749,-129.206,-101.073,164.678,58.427,160.206
C02845=1014.746,-129.456,-101.064,164.675,58.430,160.206
C02846=1014.744,-129.706,-101.053,164.673,58.433,160.206
C02847=1014.741,-129.956,-101.043,164.670,58.435,160.206
C02848=1014.740,-130.205,-101.030,164.668,58.436,160.205
C02849=1014.738,-130.455,-101.018,164.666,58.437,160.205
C02850=1014.737,-130.704,-101.006,164.664,58.438,160.204
C02851=1014.736,-130.954,-100.993,164.661,58.438,160.203
C02852=1014.736,-131.204,-100.979,164.659,58.437,160.203
C02853=1014.736,-131.454,-100.964,164.656,58.436,160.202
C02854=1014.736,-131.703,-100.949,164.655,58.434,160.201
C02855=1014.737,-131.953,-100.933,164.653,58.431,160.200
C02856=1014.738,-132.202,-100.917,164.651,58.429,160.199
C02857=1014.740,-132.452,-100.900,164.649,58.425,160.198
C02858=1014.741,-132.702,-100.883,164.646,58.422,160.196
C02859=1014.744,-132.951,-100.864,164.645,58.416,160.195
C02860=1014.747,-133.201,-100.846,164.643,58.412,160.194
C02861=1014.749,-133.451,-100.827,164.641,58.406,160.192
C02862=1014.752,-133.700,-100.807,164.639,58.400,160.190
C02863=1014.514,-133.726,-101.215,164.611,58.759,160.248
C02864=1014.510,-133.477,-101.235,164.613,58.764,160.249
C02865=1014.508,-133.227,-101.254,164.615,58.770,160.251
C02866=1014.505,-132.978,-101.273,164.617,58.775,160.252
C02867=1014.503,-132.728,-101.291,164.619,58.780,160.254
C02868=1014.501,-132.478,-101.308,164.620,58.783,160.255
C02869=1014.500,-132.229,-101.326,164.623,58.786,160.256
C02870=1014.499,-131.979,-101.342,164.625,58.789,160.257
C02871=1014.498,-131.729,-101.358,164.627,58.792,160.258
C02872=1014.498,-131.480,-101.373,164.629,58.794,160.259
C02873=1014.498,-131.229,-101.388,164.631,58.795,160.260
C02874=1014.499,-130.980,-101.401,164.633,58.795,160.261
C02875=1014.499,-130.730,-101.415,164.635,58.796,160.261
C02876=1014.500,-130.481,-101.428,164.637,58.796,160.262
C02877=1014.502,-130.231,-101.440,164.640,58.795,160.262
C02878=1014.503,-129.981,-101.451,164.642,58.793,160.263
C02879=1014.506,-129.732,-101.462,164.645,58.790,160.263
C02880=1014.507,-129.482,-101.472,164.648,58.788,160.264
C02881=1014.511,-129.233,-101.482,164.650,58.786,160.264
C02882=1014.514,-128.984,-101.491,164.652,58.782,160.264
C02883=1014.517,-128.734,-101.499,164.655,58.778,160.264
C02884=1014.521,-128.484,-101.507,164.656,58.773,160.263
C02885=1014.525,-128.234,-101.515,164.659,58.768,160.263
C02886=1014.530,-127.985,-101.522,164.662,58.762,160.263
C02887=1014.535,-127.735,-101.529,164.665,58.756,160.263
C02888=1014.539,-127.485,-101.535,164.667,58.750,160.262
C02889=1014.544,-127.236,-101.543,164.671,58.745,160.262
C02890=1014.549,-126.986,-101.549,164.673,58.739,160.262
C02891=1014.553,-126.736,-101.556,164.676,58.733,160.262
C02892=1014.558,-126.486,-101.562,164.679,58.728,160.261
C02893=1014.562,-126.237,-101.570,164.681,58.722,160.261
C02894=1014.567,-125.987,-101.576,164.683,58.716,160.261
C02895=1014.572,-125.736,-101.583,164.686,58.710,160.260
C02896=1014.577,-125.486,-101.589,164.690,58.704,160.260
C02897=1014.581,-125.237,-101.597,164.692,58.698,160.260
C02898=1014.586,-124.987,-101.603,164.694,58.692,160.259
C02899=1014.590,-124.737,-101.610,164.697,58.686,160.259
C02900=1014.595,-124.488,-101.617,164.700,58.681,160.259
C02901=1014.599,-124.238,-101.624,164.702,58.675,160.259
C02902=1014.604,-123.987,-101.632,164.704,58.669,160.258
C02903=1014.609,-123.738,-101.638,164.708,58.663,160.258
C02904=1014.613,-123.488,-101.645,164.711,58.657,160.258
C02905=1014.618,-123.238,-101.653,164.713,58.651,160.257
C02906=1014.623,-122.989,-101.659,164.716,58.646,160.257
C02907=1014.627,-122.738,-101.666,164.718,58.640,160.257
C02908=1014.632,-122.488,-101.674,164.721,58.634,160.256
C02909=1014.637,-122.239,-101.681,164.724,58.628,160.256
C02910=1014.641,-121.988,-101.687,164.727,58.623,160.256
C02911=1014.645,-121.739,-101.695,164.729,58.617,160.256
C02912=1014.650,-121.490,-101.702,164.732,58.611,160.255
C02913=1014.655,-121.239,-101.709,164.734,58.605,160.255
C02914=1014.659,-120.989,-101.716,164.738,58.598,160.255
C02915=1014.665,-120.740,-101.723,164.740,58.593,160.255
C02916=1014.669,-120.490,-101.730,164.743,58.587,160.254
C02917=1014.674,-120.240,-101.738,164.745,58.581,160.254
C02918=1014.679,-119.990,-101.744,164.748,58.575,160.253
C02919=1014.683,-119.740,-101.751,164.751,58.569,160.253
C02920=1014.687,-119.490,-101.759,164.753,58.563,160.253
C02921=1014.693,-119.240,-101.766,164.756,58.558,160.253
C02922=1014.697,-118.991,-101.773,164.759,58.552,160.252
C02923=1014.701,-118.741,-101.780,164.762,58.546,160.252
C02924=1014.707,-118.459,-101.789,164.765,58.538,160.252
C02925=1014.712,-118.177,-101.797,164.768,58.532,160.251
C02926=1014.717,-117.895,-101.805,164.771,58.525,160.251
C02927=1014.723,-117.614,-101.813,164.773,58.519,160.250
C02928=1014.728,-117.364,-101.820,164.777,58.513,160.250
C02929=1014.733,-117.114,-101.828,164.779,58.507,160.250
C02930=1014.737,-116.864,-101.835,164.782,58.501,160.249
C02931=1014.742,-116.614,-101.841,164.785,58.494,160.249
C02932=1014.747,-116.364,-101.849,164.787,58.488,160.249
C02933=1014.751,-116.114,-101.857,164.790,58.482,160.248
C02934=1014.755,-115.865,-101.864,164.793,58.476,160.248
C02935=1014.761,-115.615,-101.871,164.796,58.471,160.248
C02936=1014.765,-115.365,-101.879,164.799,58.465,160.248
C02937=1014.770,-115.115,-101.886,164.801,58.459,160.247
C02938=1014.775,-114.865,-101.894,164.804,58.453,160.247
C02939=1014.779,-114.615,-101.901,164.807,58.447,160.247
C02940=1014.785,-114.365,-101.908,164.809,58.441,160.246
C02941=1014.789,-114.116,-101.916,164.813,58.434,160.246
C02942=1014.794,-113.866,-101.923,164.815,58.428,160.246
C02943=1014.799,-113.616,-101.931,164.817,58.422,160.245
C02944=1014.803,-113.366,-101.938,164.821,58.416,160.245
C02945=1014.808,-113.116,-101.946,164.823,58.410,160.245
C02946=1014.812,-112.866,-101.953,164.825,58.404,160.244
C02947=1014.817,-112.617,-101.961,164.829,58.398,160.244
C02948=1014.822,-112.366,-101.968,164.831,58.392,160.243
C02949=1014.827,-112.117,-101.976,164.834,58.386,160.243
C02950=1014.832,-111.867,-101.984,164.837,58.380,160.243
C02951=1014.836,-111.618,-101.991,164.839,58.374,160.242
C02952=1014.841,-111.367,-101.999,164.842,58.368,160.242
C02953=1014.846,-111.118,-102.006,164.845,58.361,160.242
C02954=1014.850,-110.868,-102.014,164.848,58.355,160.241
C02955=1014.855,-110.618,-102.022,164.851,58.349,160.241
C02956=1014.860,-110.368,-102.028,164.853,58.343,160.241
C02957=1014.865,-110.119,-102.037,164.856,58.337,160.240
C02958=1014.870,-109.869,-102.044,164.859,58.331,160.240
C02959=1014.875,-109.619,-102.052,164.862,58.325,160.240
C02960=1014.879,-109.369,-102.059,164.864,58.318,160.239
C02961=1014.884,-109.119,-102.067,164.867,58.312,160.239
C02962=1014.888,-108.869,-102.075,164.869,58.306,160.238
C02963=1014.893,-108.619,-102.083,164.873,58.300,160.238
C02964=1014.898,-108.370,-102.091,164.875,58.294,160.238
C02965=1014.904,-108.120,-102.098,164.878,58.287,160.238
C02966=1014.908,-107.870,-102.105,164.881,58.281,160.237
C02967=1014.913,-107.620,-102.113,164.884,58.275,160.237
C02968=1014.918,-107.371,-102.121,164.886,58.268,160.236
C02969=1014.922,-107.120,-102.129,164.888,58.262,160.236
C02970=1014.927,-106.871,-102.136,164.892,58.256,160.236
C02971=1014.932,-106.621,-102.145,164.894,58.250,160.235
C02972=1014.936,-106.371,-102.152,164.898,58.244,160.235
C02973=1014.941,-106.121,-102.160,164.900,58.238,160.235
C02974=1014.946,-105.871,-102.169,164.902,58.232,160.234
C02975=1014.950,-105.621,-102.176,164.906,58.226,160.234
C02976=1014.955,-105.371,-102.184,164.908,58.220,160.233
C02977=1014.960,-105.122,-102.192,164.911,58.213,160.233
C02978=1014.965,-104.872,-102.200,164.914,58.207,160.233
C02979=1014.970,-104.623,-102.208,164.917,58.200,160.232
C02980=1014.974,-104.372,-102.216,164.919,58.194,160.232
C02981=1014.979,-104.122,-102.224,164.923,58.188,160.232
C02982=1014.984,-103.873,-102.232,164.925,58.182,160.231
C02983=1014.989,-103.623,-102.240,164.928,58.176,160.231
C02984=1014.994,-103.374,-102.248,164.931,58.169,160.230
C02985=1014.999,-103.123,-102.255,164.933,58.163,160.230
C02986=1015.004,-102.874,-102.264,164.936,58.157,160.230
C02987=1015.008,-102.624,-102.272,164.939,58.151,160.229
C02988=1015.013,-102.342,-102.280,164.942,58.144,160.229
C02989=1015.019,-102.061,-102.290,164.946,58.136,160.229
C02990=1015.024,-101.779,-102.298,164.948,58.129,160.228
C02991=1015.029,-101.497,-102.308,164.951,58.122,160.227
C02992=1015.034,-101.247,-102.316,164.955,58.116,160.227
C02993=1015.040,-100.997,-102.324,164.957,58.110,160.227
C02994=1015.044,-100.748,-102.332,164.960,58.103,160.226
C02995=1015.049,-100.498,-102.340,164.962,58.097,160.226
C02996=1015.054,-100.248,-102.348,164.966,58.091,160.226
C02997=1015.059,-99.999,-102.356,164.968,58.084,160.225
C02998=1015.064,-99.749,-102.365,164.971,58.078,160.225
C02999=1015.068,-99.498,-102.373,164.974,58.072,160.224
C03000=1015.074,-99.249,-102.382,164.976,58.065,160.224
C03001=1015.078,-98.999,-102.389,164.979,58.059,160.223
C03002=1015.083,-98.749,-102.397,164.982,58.052,160.223
C03003=1015.088,-98.499,-102.405,164.985,58.045,160.223
C03004=1015.093,-98.250,-102.413,164.988,58.040,160.222
C03005=1015.098,-98.000,-102.422,164.991,58.033,160.222
C03006=1015.102,-97.749,-102.430,164.993,58.027,160.221
C03007=1015.108,-97.500,-102.439,164.996,58.020,160.221
C03008=1015.112,-97.251,-102.447,164.999,58.014,160.221
C03009=1015.117,-97.001,-102.456,165.002,58.008,160.221
C03010=1015.122,-96.750,-102.464,165.005,58.002,160.220
C03011=1015.127,-96.501,-102.472,165.006,57.995,160.219
C03012=1015.132,-96.251,-102.481,165.010,57.989,160.219
C03013=1015.136,-96.002,-102.489,165.012,57.983,160.219
C03014=1015.140,-95.751,-102.498,165.016,57.977,160.219
C03015=1015.146,-95.501,-102.506,165.018,57.971,160.218
C03016=1015.151,-95.252,-102.515,165.021,57.964,160.218
C03017=1015.155,-95.002,-102.523,165.024,57.958,160.217
C03018=1015.160,-94.753,-102.532,165.027,57.952,160.217
C03019=1015.165,-94.502,-102.541,165.029,57.945,160.216
C03020=1015.170,-94.252,-102.549,165.032,57.939,160.216
C03021=1015.175,-94.002,-102.557,165.035,57.933,160.216
C03022=1015.179,-93.752,-102.566,165.038,57.927,160.215
C03023=1015.184,-93.503,-102.574,165.041,57.920,160.215
C03024=1015.189,-93.253,-102.583,165.044,57.914,160.214
C03025=1015.194,-93.004,-102.592,165.047,57.907,160.214
C03026=1015.199,-92.754,-102.600,165.049,57.901,160.213
C03027=1015.204,-92.504,-102.610,165.052,57.894,160.213
C03028=1015.209,-92.254,-102.617,165.054,57.888,160.213
C03029=1015.213,-92.005,-102.625,165.058,57.881,160.212
C03030=1015.218,-91.755,-102.634,165.060,57.876,160.212
C03031=1015.223,-91.505,-102.643,165.063,57.868,160.211
C03032=1015.228,-91.255,-102.652,165.066,57.862,160.211
C03033=1015.233,-91.005,-102.661,165.068,57.856,160.210
C03034=1015.238,-90.755,-102.669,165.072,57.849,160.210
C03035=1015.243,-90.505,-102.678,165.074,57.843,160.210
C03036=1015.248,-90.256,-102.687,165.077,57.836,160.209
C03037=1015.253,-90.006,-102.696,165.081,57.830,160.209
C03038=1015.257,-89.757,-102.704,165.082,57.823,160.208
C03039=1015.262,-89.507,-102.712,165.086,57.817,160.208
C03040=1015.267,-89.257,-102.721,165.089,57.810,160.208
C03041=1015.272,-89.007,-102.730,165.091,57.804,160.207
C03042=1015.277,-88.757,-102.739,165.094,57.797,160.207
C03043=1015.282,-88.507,-102.747,165.097,57.791,160.206
C03044=1015.287,-88.257,-102.756,165.099,57.784,160.206
C03045=1015.292,-88.008,-102.765,165.103,57.778,160.206
C03046=1015.297,-87.758,-102.773,165.105,57.771,160.205
C03047=1015.302,-87.508,-102.783,165.108,57.765,160.205
C03048=1015.307,-87.258,-102.791,165.111,57.758,160.204
C03049=1015.311,-87.008,-102.800,165.113,57.751,160.203
C03050=1015.317,-86.758,-102.809,165.117,57.745,160.203
C03051=1015.322,-86.509,-102.817,165.119,57.738,160.203
C03052=1015.328,-86.230,-102.827,165.122,57.731,160.202
C03053=1015.333,-85.950,-102.837,165.125,57.724,160.202
C03054=1015.339,-85.670,-102.847,165.129,57.716,160.201
C03055=1015.345,-85.391,-102.857,165.132,57.709,160.200
C03056=1015.349,-85.141,-102.866,165.135,57.702,160.200
C03057=1015.354,-84.891,-102.875,165.138,57.695,160.200
C03058=1015.359,-84.641,-102.884,165.140,57.689,160.199
C03059=1015.364,-84.391,-102.892,165.143,57.682,160.199
C03060=1015.369,-84.141,-102.901,165.146,57.675,160.198
C03061=1015.374,-83.891,-102.910,165.149,57.668,160.198
C03062=1015.379,-83.642,-102.918,165.152,57.662,160.197
C03063=1015.384,-83.392,-102.928,165.155,57.655,160.197
C03064=1015.390,-83.099,-102.938,165.158,57.647,160.196
C03065=1015.396,-82.805,-102.949,165.161,57.639,160.196
C03066=1015.402,-82.512,-102.959,165.164,57.632,160.195
C03067=1015.408,-82.218,-102.969,165.168,57.624,160.195
C03068=1015.413,-81.968,-102.978,165.171,57.617,160.194
C03069=1015.418,-81.718,-102.987,165.174,57.610,160.193
C03070=1015.423,-81.468,-102.996,165.176,57.604,160.193
C03071=1015.428,-81.218,-103.006,165.179,57.597,160.193
C03072=1015.433,-80.969,-103.014,165.182,57.590,160.192
C03073=1015.439,-80.719,-103.022,165.185,57.583,160.192
C03074=1015.443,-80.469,-103.032,165.188,57.576,160.191
C03075=1015.448,-80.220,-103.041,165.190,57.570,160.191
C03076=1015.453,-79.970,-103.050,165.193,57.563,160.190
C03077=1015.458,-79.719,-103.059,165.197,57.557,160.190
C03078=1015.463,-79.470,-103.069,165.199,57.550,160.189
C03079=1015.468,-79.220,-103.078,165.202,57.543,160.189
C03080=1015.473,-78.971,-103.087,165.205,57.537,160.188
C03081=1015.478,-78.721,-103.096,165.207,57.530,160.188
C03082=1015.483,-78.472,-103.106,165.210,57.523,160.187
C03083=1015.488,-78.221,-103.115,165.213,57.517,160.187
C03084=1015.493,-77.971,-103.124,165.216,57.510,160.186
C03085=1015.498,-77.721,-103.134,165.218,57.503,160.186
C03086=1015.503,-77.472,-103.142,165.222,57.497,160.185
C03087=1015.508,-77.222,-103.152,165.225,57.490,160.185
C03088=1015.512,-76.972,-103.161,165.227,57.483,160.184
C03089=1015.519,-76.722,-103.171,165.230,57.477,160.184
C03090=1015.523,-76.472,-103.180,165.233,57.470,160.183
C03091=1015.528,-76.223,-103.190,165.236,57.463,160.183
C03092=1015.533,-75.973,-103.198,165.238,57.457,160.182
C03093=1015.538,-75.724,-103.208,165.241,57.450,160.182
C03094=1015.543,-75.473,-103.218,165.244,57.443,160.181
C03095=1015.548,-75.224,-103.227,165.247,57.436,160.181
C03096=1015.553,-74.974,-103.236,165.249,57.430,160.180
C03097=1015.558,-74.725,-103.246,165.253,57.423,160.180
C03098=1015.564,-74.474,-103.256,165.256,57.416,160.180
C03099=1015.568,-74.224,-103.265,165.258,57.410,160.179
C03100=1015.573,-73.975,-103.275,165.261,57.404,160.179
C03101=1015.578,-73.726,-103.284,165.264,57.397,160.178
C03102=1015.583,-73.475,-103.294,165.266,57.391,160.178
C03103=1015.588,-73.226,-103.304,165.269,57.384,160.177
C03104=1015.593,-72.976,-103.313,165.272,57.377,160.177
C03105=1015.598,-72.726,-103.324,165.275,57.371,160.176
C03106=1015.603,-72.476,-103.333,165.278,57.364,160.176
C03107=1015.607,-72.227,-103.342,165.281,57.358,160.175
C03108=1015.612,-71.977,-103.352,165.283,57.351,160.175
C03109=1015.618,-71.727,-103.362,165.286,57.344,160.174
C03110=1015.622,-71.478,-103.372,165.290,57.338,160.174
C03111=1015.627,-71.228,-103.381,165.292,57.331,160.173
C03112=1015.633,-70.986,-103.391,165.295,57.325,160.173
C03113=1015.637,-70.744,-103.400,165.297,57.318,160.172
C03114=1015.642,-70.502,-103.410,165.301,57.312,160.172
C03115=1015.646,-70.261,-103.420,165.303,57.306,160.171
C03116=1015.651,-70.019,-103.429,165.306,57.299,160.171
C03117=1015.656,-69.777,-103.439,165.308,57.293,160.170
C03118=1015.661,-69.535,-103.448,165.311,57.286,160.170
C03119=1015.666,-69.294,-103.458,165.313,57.280,160.169
C03120=1015.671,-69.044,-103.467,165.316,57.273,160.169
C03121=1015.676,-68.795,-103.477,165.319,57.266,160.168
C03122=1015.681,-68.545,-103.487,165.322,57.260,160.168
C03123=1015.686,-68.295,-103.496,165.325,57.253,160.167
C03124=1015.690,-68.044,-103.507,165.328,57.246,160.167
C03125=1015.695,-67.795,-103.517,165.331,57.239,160.166
C03126=1015.700,-67.545,-103.527,165.333,57.233,160.166
C03127=1015.706,-67.295,-103.537,165.336,57.226,160.165
C03128=1015.710,-67.046,-103.547,165.339,57.219,160.165
C03129=1015.715,-66.796,-103.556,165.342,57.212,160.164
C03130=1015.721,-66.546,-103.567,165.344,57.206,160.164
C03131=1015.726,-66.297,-103.576,165.347,57.199,160.163
C03132=1015.731,-66.047,-103.587,165.351,57.193,160.163
C03133=1015.736,-65.797,-103.596,165.354,57.186,160.162
C03134=1015.741,-65.547,-103.607,165.356,57.179,160.162
C03135=1015.746,-65.298,-103.616,165.359,57.172,160.161
C03136=1015.751,-65.048,-103.626,165.362,57.165,160.161
C03137=1015.756,-64.798,-103.636,165.364,57.158,160.160
C03138=1015.761,-64.549,-103.646,165.366,57.152,160.159
C03139=1015.767,-64.299,-103.656,165.369,57.145,160.159
C03140=1015.771,-64.049,-103.666,165.373,57.139,160.159
C03141=1015.777,-63.799,-103.676,165.376,57.132,160.158
C03142=1015.782,-63.550,-103.686,165.379,57.125,160.158
C03143=1015.787,-63.300,-103.696,165.381,57.118,160.157
C03144=1015.792,-63.050,-103.706,165.384,57.111,160.156
C03145=1015.797,-62.800,-103.716,165.387,57.104,160.156
C03146=1015.802,-62.551,-103.726,165.390,57.097,160.155
C03147=1015.808,-62.301,-103.736,165.393,57.090,160.155
C03148=1015.812,-62.051,-103.746,165.395,57.084,160.154
C03149=1015.818,-61.801,-103.756,165.398,57.077,160.154
C03150=1015.823,-61.552,-103.766,165.401,57.070,160.153
C03151=1015.828,-61.302,-103.776,165.404,57.063,160.153
C03152=1015.833,-61.052,-103.786,165.407,57.056,160.152
C03153=1015.838,-60.802,-103.796,165.410,57.049,160.151
C03154=1015.843,-60.553,-103.806,165.412,57.042,160.151
C03155=1015.848,-60.302,-103.816,165.415,57.035,160.150
C03156=1015.853,-60.053,-103.826,165.418,57.028,160.150
C03157=1015.859,-59.804,-103.837,165.421,57.021,160.149
C03158=1015.864,-59.553,-103.847,165.424,57.014,160.149
C03159=1015.869,-59.304,-103.857,165.427,57.007,160.148
C03160=1015.874,-59.054,-103.867,165.430,57.001,160.148
C03161=1015.879,-58.804,-103.877,165.432,56.993,160.147
C03162=1015.885,-58.554,-103.887,165.434,56.986,160.146
C03163=1015.889,-58.305,-103.897,165.437,56.979,160.146
C03164=1015.895,-58.055,-103.908,165.440,56.972,160.145
C03165=1015.901,-57.805,-103.918,165.443,56.965,160.145
C03166=1015.905,-57.556,-103.928,165.446,56.959,160.144
C03167=1015.911,-57.306,-103.938,165.449,56.952,160.143
C03168=1015.916,-57.056,-103.948,165.452,56.945,160.143
C03169=1015.921,-56.807,-103.959,165.455,56.937,160.142
C03170=1015.927,-56.557,-103.969,165.458,56.930,160.142
C03171=1015.932,-56.307,-103.979,165.460,56.923,160.141
C03172=1015.937,-56.057,-103.989,165.463,56.917,160.140
C03173=1015.942,-55.807,-104.000,165.466,56.910,160.140
C03174=1015.947,-55.558,-104.010,165.468,56.902,160.139
C03175=1015.952,-55.308,-104.020,165.471,56.895,160.139
C03176=1015.958,-55.058,-104.030,165.474,56.888,160.138
C03177=1015.963,-54.809,-104.041,165.477,56.881,160.138
C03178=1015.968,-54.559,-104.051,165.480,56.874,160.137
C03179=1015.974,-54.309,-104.061,165.483,56.866,160.136
C03180=1015.979,-54.032,-104.072,165.485,56.859,160.135
C03181=1015.986,-53.756,-104.084,165.489,56.851,160.135
C03182=1015.991,-53.480,-104.095,165.493,56.843,160.134
C03183=1015.997,-53.203,-104.107,165.495,56.836,160.134
C03184=1016.002,-52.954,-104.117,165.498,56.828,160.133
C03185=1016.008,-52.703,-104.127,165.501,56.821,160.132
C03186=1016.013,-52.454,-104.138,165.504,56.814,160.132
C03187=1016.019,-52.204,-104.148,165.506,56.806,160.131
C03188=1016.024,-51.954,-104.158,165.509,56.800,160.130
C03189=1016.029,-51.705,-104.169,165.512,56.793,160.130
C03190=1016.035,-51.455,-104.179,165.515,56.785,160.129
C03191=1016.039,-51.205,-104.189,165.518,56.778,160.129
C03192=1016.045,-50.956,-104.200,165.521,56.771,160.128
C03193=1016.050,-50.706,-104.210,165.524,56.764,160.128
C03194=1016.055,-50.456,-104.222,165.526,56.758,160.127
C03195=1016.060,-50.206,-104.232,165.529,56.751,160.126
C03196=1016.065,-49.956,-104.243,165.532,56.744,160.126
C03197=1016.071,-49.707,-104.254,165.535,56.737,160.125
C03198=1016.075,-49.457,-104.265,165.538,56.730,160.125
C03199=1016.081,-49.207,-104.275,165.540,56.723,160.124
C03200=1016.086,-48.957,-104.287,165.542,56.716,160.123
C03201=1016.091,-48.708,-104.297,165.545,56.709,160.123
///RCONF 1,0,0,0,0,0,0,0,0,0,0,0,0,0,0,0,0,0,0,0,0,0,0,0
C03202=1016.096,-48.458,-104.308,165.548,56.702,160.122
C03203=1016.101,-48.208,-104.318,165.551,56.695,160.122
C03204=1016.106,-47.958,-104.330,165.555,56.688,160.121
C03205=1016.112,-47.709,-104.341,165.556,56.682,160.120
C03206=1016.116,-47.459,-104.351,165.560,56.675,160.120
C03207=1016.122,-47.209,-104.362,165.563,56.668,160.119
C03208=1016.127,-46.960,-104.373,165.565,56.660,160.119
C03209=1016.132,-46.710,-104.384,165.568,56.653,160.118
C03210=1016.137,-46.460,-104.395,165.571,56.646,160.118
C03211=1016.142,-46.211,-104.406,165.573,56.640,160.117
C03212=1016.147,-45.961,-104.417,165.576,56.633,160.116
C03213=1016.153,-45.711,-104.427,165.579,56.625,160.115
C03214=1016.158,-45.461,-104.439,165.582,56.618,160.115
C03215=1016.164,-45.212,-104.450,165.585,56.611,160.114
C03216=1016.169,-44.962,-104.460,165.588,56.605,160.114
C03217=1016.174,-44.712,-104.471,165.591,56.598,160.113
C03218=1016.179,-44.463,-104.482,165.592,56.590,160.112
C03219=1016.184,-44.213,-104.493,165.595,56.584,160.112
C03220=1016.190,-43.964,-104.504,165.599,56.577,160.111
C03221=1016.195,-43.713,-104.515,165.602,56.570,160.111
C03222=1016.200,-43.464,-104.526,165.604,56.562,160.110
C03223=1016.205,-43.214,-104.537,165.607,56.555,160.109
C03224=1016.211,-42.965,-104.548,165.610,56.548,160.109
C03225=1016.216,-42.714,-104.559,165.613,56.541,160.108
C03226=1016.221,-42.465,-104.570,165.616,56.534,160.108
C03227=1016.226,-42.215,-104.581,165.618,56.527,160.107
C03228=1016.232,-41.966,-104.592,165.621,56.520,160.106
C03229=1016.237,-41.716,-104.603,165.623,56.513,160.106
C03230=1016.242,-41.467,-104.614,165.626,56.506,160.105
C03231=1016.247,-41.216,-104.625,165.629,56.499,160.105
C03232=1016.253,-40.967,-104.636,165.632,56.491,160.104
C03233=1016.258,-40.717,-104.647,165.635,56.484,160.103
C03234=1016.264,-40.468,-104.658,165.638,56.477,160.102
C03235=1016.269,-40.218,-104.670,165.641,56.470,160.102
C03236=1016.274,-39.968,-104.680,165.644,56.463,160.101
C03237=1016.279,-39.719,-104.692,165.646,56.455,160.101
C03238=1016.285,-39.468,-104.702,165.649,56.449,160.100
C03239=1016.290,-39.219,-104.713,165.651,56.442,160.099
C03240=1016.295,-38.969,-104.725,165.654,56.435,160.099
C03241=1016.300,-38.719,-104.736,165.657,56.428,160.098
C03242=1016.306,-38.470,-104.748,165.660,56.421,160.097
C03243=1016.311,-38.220,-104.759,165.663,56.414,160.097
C03244=1016.316,-37.943,-104.772,165.666,56.406,160.096
C03245=1016.322,-37.668,-104.784,165.668,56.399,160.095
C03246=1016.327,-37.391,-104.797,165.672,56.391,160.095
C03247=1016.334,-37.115,-104.810,165.674,56.383,160.094
C03248=1016.339,-36.865,-104.822,165.677,56.376,160.093
C03249=1016.344,-36.616,-104.833,165.680,56.369,160.093
C03250=1016.350,-36.366,-104.844,165.683,56.362,160.092
C03251=1016.355,-36.116,-104.856,165.686,56.355,160.092
C03252=1016.360,-35.867,-104.867,165.689,56.348,160.091
C03253=1016.365,-35.617,-104.878,165.691,56.341,160.090
C03254=1016.370,-35.367,-104.889,165.694,56.334,160.089
C03255=1016.375,-35.117,-104.901,165.697,56.327,160.089
C03256=1016.380,-34.868,-104.912,165.700,56.320,160.088
C03257=1016.386,-34.618,-104.924,165.703,56.312,160.088
C03258=1016.391,-34.369,-104.935,165.706,56.306,160.087
C03259=1016.396,-34.119,-104.947,165.709,56.299,160.087
C03260=1016.401,-33.869,-104.958,165.710,56.292,160.086
C03261=1016.406,-33.620,-104.970,165.713,56.285,160.085
C03262=1016.412,-33.370,-104.982,165.716,56.277,160.084
C03263=1016.417,-33.121,-104.993,165.719,56.270,160.084
C03264=1016.423,-32.870,-105.005,165.722,56.263,160.083
C03265=1016.428,-32.621,-105.016,165.725,56.256,160.082
C03266=1016.433,-32.371,-105.028,165.728,56.249,160.082
C03267=1016.438,-32.122,-105.040,165.730,56.241,160.081
C03268=1016.444,-31.872,-105.051,165.733,56.234,160.081
C03269=1016.449,-31.622,-105.062,165.735,56.228,160.080
C03270=1016.454,-31.373,-105.074,165.738,56.220,160.079
C03271=1016.459,-31.123,-105.085,165.741,56.214,160.078
C03272=1016.465,-30.874,-105.097,165.744,56.206,160.078
C03273=1016.471,-30.623,-105.109,165.747,56.199,160.077
C03274=1016.476,-30.374,-105.120,165.749,56.191,160.076
C03275=1016.481,-30.124,-105.132,165.752,56.185,160.076
C03276=1016.486,-29.875,-105.144,165.755,56.177,160.075
C03277=1016.492,-29.625,-105.155,165.758,56.170,160.075
C03278=1016.497,-29.375,-105.166,165.761,56.163,160.074
C03279=1016.503,-29.125,-105.179,165.764,56.156,160.073
C03280=1016.508,-28.876,-105.190,165.765,56.149,160.072
C03281=1016.513,-28.626,-105.202,165.768,56.142,160.072
C03282=1016.519,-28.377,-105.213,165.771,56.134,160.071
C03283=1016.524,-28.127,-105.225,165.774,56.127,160.070
C03284=1016.529,-27.877,-105.236,165.777,56.120,160.070
C03285=1016.535,-27.627,-105.249,165.780,56.113,160.069
C03286=1016.540,-27.378,-105.260,165.782,56.105,160.068
C03287=1016.545,-27.128,-105.272,165.785,56.098,160.068
C03288=1016.551,-26.878,-105.284,165.789,56.092,160.067
C03289=1016.556,-26.629,-105.296,165.790,56.084,160.066
C03290=1016.561,-26.379,-105.308,165.793,56.078,160.066
C03291=1016.566,-26.130,-105.320,165.796,56.071,160.065
C03292=1016.571,-25.880,-105.331,165.799,56.063,160.064
C03293=1016.577,-25.630,-105.344,165.802,56.056,160.064
C03294=1016.581,-25.380,-105.356,165.804,56.049,160.063
C03295=1016.587,-25.131,-105.368,165.807,56.042,160.062
C03296=1016.592,-24.881,-105.380,165.809,56.035,160.061
C03297=1016.598,-24.631,-105.392,165.812,56.028,160.061
C03298=1016.603,-24.381,-105.404,165.816,56.021,160.060
C03299=1016.608,-24.132,-105.416,165.818,56.014,160.060
C03300=1016.613,-23.883,-105.428,165.820,56.007,160.059
C03301=1016.619,-23.632,-105.440,165.823,56.000,160.058
C03302=1016.624,-23.383,-105.452,165.826,55.993,160.058
C03303=1016.629,-23.133,-105.464,165.829,55.985,160.057
C03304=1016.634,-22.884,-105.476,165.832,55.978,160.056
C03305=1016.640,-22.634,-105.488,165.834,55.971,160.055
C03306=1016.645,-22.385,-105.500,165.837,55.964,160.055
C03307=1016.650,-22.135,-105.513,165.839,55.957,160.054
C03308=1016.656,-21.858,-105.526,165.843,55.949,160.053
C03309=1016.662,-21.580,-105.539,165.846,55.941,160.053
C03310=1016.668,-21.303,-105.553,165.849,55.933,160.052
C03311=1016.675,-21.026,-105.566,165.852,55.925,160.051
C03312=1016.680,-20.776,-105.578,165.854,55.918,160.050
C03313=1016.685,-20.527,-105.590,165.857,55.911,160.050
C03314=1016.691,-20.277,-105.603,165.860,55.904,160.049
C03315=1016.695,-20.027,-105.615,165.863,55.896,160.048
C03316=1016.700,-19.778,-105.627,165.866,55.890,160.048
C03317=1016.706,-19.528,-105.639,165.868,55.882,160.047
C03318=1016.711,-19.278,-105.651,165.871,55.874,160.046
C03319=1016.717,-19.029,-105.663,165.874,55.868,160.046
C03320=1016.722,-18.779,-105.676,165.877,55.860,160.045
C03321=1016.728,-18.530,-105.688,165.879,55.854,160.044
C03322=1016.733,-18.280,-105.699,165.881,55.846,160.043
C03323=1016.739,-18.030,-105.712,165.884,55.839,160.042
C03324=1016.744,-17.781,-105.724,165.887,55.832,160.042
C03325=1016.750,-17.530,-105.736,165.890,55.824,160.041
C03326=1016.754,-17.281,-105.749,165.892,55.817,160.040
C03327=1016.759,-17.032,-105.761,165.896,55.810,160.040
C03328=1016.765,-16.782,-105.773,165.898,55.802,160.039
C03329=1016.770,-16.532,-105.785,165.901,55.795,160.038
C03330=1016.776,-16.282,-105.797,165.904,55.788,160.038
C03331=1016.782,-16.033,-105.810,165.907,55.780,160.037
C03332=1016.787,-15.784,-105.822,165.909,55.774,160.036
C03333=1016.792,-15.534,-105.835,165.911,55.767,160.035
C03334=1016.797,-15.284,-105.847,165.915,55.760,160.035
C03335=1016.803,-15.035,-105.860,165.917,55.752,160.034
C03336=1016.808,-14.785,-105.872,165.920,55.745,160.033
C03337=1016.814,-14.535,-105.885,165.922,55.738,160.033
C03338=1016.818,-14.286,-105.898,165.925,55.731,160.032
C03339=1016.824,-14.036,-105.910,165.928,55.724,160.031
C03340=1016.830,-13.787,-105.922,165.931,55.717,160.031
C03341=1016.834,-13.537,-105.935,165.934,55.710,160.030
C03342=1016.840,-13.287,-105.948,165.936,55.702,160.029
C03343=1016.845,-13.038,-105.960,165.938,55.696,160.028
C03344=1016.851,-12.788,-105.973,165.941,55.688,160.028
C03345=1016.856,-12.539,-105.985,165.944,55.681,160.027
C03346=1016.861,-12.288,-105.999,165.947,55.674,160.026
C03347=1016.866,-12.039,-106.011,165.950,55.667,160.026
C03348=1016.872,-11.789,-106.023,165.953,55.660,160.025
C03349=1016.877,-11.540,-106.036,165.954,55.652,160.024
C03350=1016.883,-11.290,-106.049,165.957,55.646,160.023
C03351=1016.888,-11.041,-106.061,165.960,55.638,160.023
C03352=1016.893,-10.791,-106.074,165.963,55.631,160.022
C03353=1016.898,-10.541,-106.086,165.966,55.624,160.021
C03354=1016.904,-10.291,-106.099,165.968,55.616,160.020
C03355=1016.909,-10.042,-106.111,165.972,55.610,160.020
C03356=1016.915,-9.792,-106.124,165.973,55.602,160.019
C03357=1016.919,-9.543,-106.137,165.976,55.595,160.018
C03358=1016.925,-9.293,-106.149,165.979,55.588,160.018
C03359=1016.931,-9.044,-106.162,165.982,55.581,160.017
C03360=1016.936,-8.793,-106.175,165.984,55.573,160.016
C03361=1016.941,-8.544,-106.187,165.988,55.566,160.016
C03362=1016.947,-8.295,-106.201,165.990,55.559,160.015
C03363=1016.953,-8.045,-106.213,165.992,55.552,160.014
C03364=1016.958,-7.796,-106.225,165.995,55.544,160.013
C03365=1016.963,-7.545,-106.239,165.998,55.538,160.012
C03366=1016.968,-7.296,-106.251,166.000,55.530,160.012
C03367=1016.973,-7.046,-106.264,166.003,55.523,160.011
C03368=1016.979,-6.797,-106.276,166.006,55.515,160.010
C03369=1016.985,-6.548,-106.289,166.009,55.508,160.010
C03370=1016.990,-6.297,-106.303,166.012,55.501,160.009
C03371=1016.995,-6.048,-106.315,166.014,55.493,160.008
C03372=1017.002,-5.769,-106.329,166.017,55.486,160.007
C03373=1017.008,-5.490,-106.343,166.020,55.477,160.006
C03374=1017.014,-5.211,-106.358,166.022,55.469,160.005
C03375=1017.019,-4.932,-106.372,166.026,55.461,160.005
C03376=1017.025,-4.682,-106.385,166.029,55.454,160.004
C03377=1017.031,-4.432,-106.397,166.032,55.446,160.003
C03378=1017.036,-4.183,-106.411,166.035,55.439,160.002
C03379=1017.041,-3.933,-106.424,166.036,55.432,160.001
C03380=1017.046,-3.683,-106.437,166.040,55.425,160.001
C03381=1017.052,-3.434,-106.450,166.042,55.418,160.000
C03382=1017.057,-3.184,-106.463,166.045,55.410,159.999
C03383=1017.062,-2.935,-106.477,166.047,55.404,159.999
C03384=1017.067,-2.685,-106.490,166.050,55.397,159.998
C03385=1017.073,-2.435,-106.502,166.053,55.390,159.997
C03386=1017.078,-2.186,-106.516,166.056,55.382,159.997
C03387=1017.083,-1.936,-106.529,166.058,55.376,159.996
C03388=1017.089,-1.686,-106.543,166.061,55.369,159.995
C03389=1017.094,-1.437,-106.555,166.063,55.361,159.994
C03390=1017.099,-1.188,-106.569,166.066,55.354,159.994
C03391=1017.105,-0.938,-106.582,166.068,55.347,159.993
C03392=1017.110,-0.689,-106.596,166.071,55.340,159.992
C03393=1017.115,-0.439,-106.608,166.074,55.333,159.991
C03394=1017.121,-0.189,-106.622,166.077,55.326,159.991
C03395=1017.126,0.061,-106.635,166.080,55.319,159.990
C03396=1017.131,0.310,-106.649,166.082,55.312,159.989
C03397=1017.136,0.560,-106.662,166.084,55.304,159.988
C03398=1017.142,0.809,-106.675,166.088,55.298,159.988
C03399=1017.147,1.059,-106.688,166.090,55.290,159.987
C03400=1017.152,1.308,-106.702,166.092,55.283,159.986
C03401=1017.158,1.559,-106.715,166.095,55.276,159.985
C03402=1017.163,1.807,-106.728,166.098,55.269,159.985
C03403=1017.168,2.057,-106.741,166.101,55.261,159.984
C03404=1017.174,2.307,-106.755,166.103,55.254,159.983
C03405=1017.179,2.556,-106.769,166.105,55.248,159.982
C03406=1017.185,2.806,-106.781,166.108,55.240,159.982
C03407=1017.190,3.055,-106.795,166.111,55.233,159.981
C03408=1017.195,3.305,-106.808,166.114,55.225,159.980
C03409=1017.201,3.555,-106.822,166.117,55.218,159.980
C03410=1017.206,3.804,-106.835,166.118,55.211,159.979
C03411=1017.211,4.054,-106.848,166.121,55.204,159.978
C03412=1017.217,4.303,-106.862,166.124,55.196,159.977
C03413=1017.222,4.554,-106.875,166.127,55.190,159.976
C03414=1017.228,4.803,-106.889,166.130,55.182,159.976
C03415=1017.233,5.052,-106.902,166.133,55.175,159.975
C03416=1017.238,5.302,-106.915,166.134,55.168,159.974
C03417=1017.244,5.551,-106.929,166.137,55.160,159.973
C03418=1017.249,5.801,-106.942,166.140,55.153,159.972
C03419=1017.255,6.050,-106.955,166.143,55.146,159.972
C03420=1017.260,6.300,-106.968,166.146,55.139,159.971
C03421=1017.265,6.550,-106.982,166.148,55.131,159.970
C03422=1017.271,6.800,-106.996,166.150,55.124,159.969
C03423=1017.276,7.049,-107.009,166.153,55.117,159.968
C03424=1017.282,7.298,-107.023,166.156,55.109,159.968
C03425=1017.287,7.548,-107.035,166.159,55.103,159.967
C03426=1017.292,7.797,-107.049,166.162,55.095,159.966
C03427=1017.298,8.047,-107.063,166.164,55.088,159.966
C03428=1017.303,8.297,-107.076,166.167,55.080,159.965
C03429=1017.309,8.546,-107.090,166.169,55.073,159.964
C03430=1017.315,8.796,-107.103,166.172,55.066,159.963
C03431=1017.319,9.046,-107.116,166.174,55.058,159.962
C03432=1017.325,9.295,-107.130,166.177,55.051,159.961
C03433=1017.331,9.544,-107.143,166.180,55.043,159.961
C03434=1017.337,9.794,-107.157,166.183,55.036,159.960
C03435=1017.342,10.044,-107.170,166.186,55.029,159.959
C03436=1017.348,10.325,-107.186,166.188,55.021,159.958
C03437=1017.355,10.606,-107.201,166.191,55.013,159.957
C03438=1017.360,10.887,-107.217,166.194,55.004,159.956
C03439=1017.366,11.168,-107.231,166.197,54.996,159.955
C03440=1017.372,11.418,-107.245,166.200,54.988,159.955
C03441=1017.377,11.667,-107.259,166.202,54.981,159.954
C03442=1017.383,11.916,-107.272,166.205,54.974,159.953
C03443=1017.389,12.167,-107.286,166.208,54.966,159.952
C03444=1017.394,12.416,-107.299,166.210,54.959,159.951
C03445=1017.400,12.666,-107.313,166.212,54.952,159.951
C03446=1017.406,12.915,-107.327,166.215,54.944,159.950
C03447=1017.411,13.165,-107.340,166.218,54.937,159.949
C03448=1017.417,13.414,-107.354,166.221,54.929,159.948
C03449=1017.422,13.664,-107.368,166.224,54.923,159.948
C03450=1017.427,13.914,-107.382,166.226,54.916,159.947
C03451=1017.432,14.164,-107.396,166.228,54.908,159.946
C03452=1017.437,14.413,-107.409,166.231,54.901,159.945
C03453=1017.442,14.662,-107.423,166.234,54.894,159.944
C03454=1017.448,14.912,-107.437,166.237,54.886,159.944
C03455=1017.453,15.161,-107.451,166.239,54.880,159.943
C03456=1017.459,15.411,-107.465,166.242,54.872,159.942
C03457=1017.464,15.661,-107.479,166.245,54.865,159.941
C03458=1017.470,15.910,-107.492,166.247,54.858,159.940
C03459=1017.476,16.159,-107.507,166.250,54.850,159.940
C03460=1017.481,16.409,-107.521,166.252,54.843,159.939
C03461=1017.487,16.658,-107.535,166.255,54.836,159.938
C03462=1017.491,16.908,-107.549,166.257,54.828,159.937
C03463=1017.497,17.158,-107.563,166.261,54.822,159.937
C03464=1017.502,17.407,-107.577,166.263,54.814,159.936
C03465=1017.508,17.657,-107.591,166.265,54.807,159.935
C03466=1017.513,17.906,-107.605,166.268,54.800,159.934
C03467=1017.519,18.156,-107.619,166.271,54.792,159.933
C03468=1017.524,18.406,-107.632,166.274,54.785,159.933
C03469=1017.530,18.655,-107.646,166.276,54.778,159.932
C03470=1017.535,18.905,-107.660,166.278,54.771,159.931
C03471=1017.541,19.154,-107.674,166.281,54.763,159.930
C03472=1017.546,19.404,-107.689,166.284,54.756,159.929
C03473=1017.551,19.653,-107.703,166.287,54.748,159.928
C03474=1017.557,19.903,-107.717,166.289,54.742,159.928
C03475=1017.562,20.152,-107.731,166.292,54.735,159.927
C03476=1017.567,20.402,-107.745,166.294,54.727,159.926
C03477=1017.573,20.651,-107.760,166.297,54.720,159.925
C03478=1017.578,20.901,-107.774,166.299,54.713,159.924
C03479=1017.584,21.150,-107.787,166.302,54.706,159.924
C03480=1017.588,21.400,-107.802,166.305,54.698,159.923
C03481=1017.594,21.649,-107.817,166.307,54.691,159.922
C03482=1017.600,21.899,-107.830,166.310,54.683,159.921
C03483=1017.606,22.149,-107.845,166.312,54.676,159.920
C03484=1017.611,22.399,-107.858,166.315,54.669,159.920
C03485=1017.616,22.648,-107.874,166.318,54.662,159.919
C03486=1017.622,22.897,-107.888,166.321,54.655,159.918
C03487=1017.627,23.147,-107.901,166.323,54.648,159.917
C03488=1017.633,23.397,-107.915,166.325,54.641,159.916
C03489=1017.638,23.646,-107.930,166.328,54.633,159.916
C03490=1017.643,23.895,-107.944,166.331,54.626,159.915
C03491=1017.649,24.145,-107.958,166.334,54.618,159.914
C03492=1017.654,24.394,-107.973,166.336,54.611,159.913
C03493=1017.659,24.644,-107.987,166.338,54.604,159.912
C03494=1017.665,24.893,-108.001,166.341,54.597,159.912
C03495=1017.671,25.143,-108.016,166.344,54.589,159.911
C03496=1017.676,25.393,-108.030,166.347,54.582,159.910
C03497=1017.681,25.643,-108.044,166.349,54.575,159.909
C03498=1017.687,25.891,-108.059,166.351,54.568,159.908
C03499=1017.692,26.141,-108.073,166.354,54.560,159.907
C03500=1017.698,26.424,-108.089,166.358,54.552,159.907
C03501=1017.705,26.706,-108.106,166.360,54.544,159.906
C03502=1017.711,26.988,-108.122,166.363,54.535,159.905
C03503=1017.717,27.271,-108.138,166.366,54.527,159.904
C03504=1017.722,27.520,-108.153,166.369,54.520,159.903
C03505=1017.727,27.770,-108.167,166.371,54.512,159.902
C03506=1017.733,28.020,-108.182,166.373,54.505,159.901
C03507=1017.738,28.270,-108.197,166.376,54.498,159.900
C03508=1017.744,28.519,-108.211,166.379,54.491,159.900
C03509=1017.749,28.768,-108.225,166.382,54.484,159.899
C03510=1017.755,29.018,-108.240,166.384,54.477,159.898
C03511=1017.760,29.267,-108.254,166.387,54.470,159.897
C03512=1017.766,29.517,-108.270,166.390,54.462,159.897
C03513=1017.771,29.767,-108.284,166.393,54.455,159.896
C03514=1017.776,30.016,-108.299,166.394,54.448,159.895
C03515=1017.782,30.266,-108.313,166.397,54.441,159.894
C03516=1017.787,30.515,-108.328,166.400,54.433,159.893
C03517=1017.793,30.765,-108.342,166.403,54.426,159.892
C03518=1017.798,31.014,-108.357,166.405,54.419,159.891
C03519=1017.804,31.263,-108.372,166.408,54.412,159.891
C03520=1017.808,31.513,-108.386,166.410,54.404,159.890
C03521=1017.814,31.762,-108.401,166.413,54.397,159.889
C03522=1017.819,32.013,-108.416,166.415,54.390,159.888
C03523=1017.825,32.262,-108.430,166.418,54.383,159.887
C03524=1017.830,32.511,-108.445,166.421,54.375,159.887
C03525=1017.836,32.761,-108.459,166.424,54.368,159.886
C03526=1017.841,33.010,-108.474,166.425,54.361,159.885
C03527=1017.847,33.259,-108.489,166.428,54.354,159.884
C03528=1017.852,33.509,-108.504,166.431,54.346,159.883
C03529=1017.858,33.758,-108.518,166.434,54.339,159.883
C03530=1017.862,34.008,-108.533,166.436,54.332,159.882
C03531=1017.869,34.258,-108.548,166.439,54.325,159.881
C03532=1017.874,34.507,-108.563,166.442,54.317,159.880
C03533=1017.879,34.757,-108.577,166.444,54.310,159.879
C03534=1017.884,35.006,-108.592,166.447,54.303,159.878
C03535=1017.891,35.256,-108.607,166.449,54.295,159.877
C03536=1017.896,35.505,-108.622,166.451,54.288,159.876
C03537=1017.901,35.754,-108.636,166.454,54.280,159.876
C03538=1017.907,36.004,-108.652,166.457,54.273,159.875
C03539=1017.912,36.254,-108.667,166.459,54.266,159.874
C03540=1017.917,36.503,-108.681,166.462,54.259,159.873
C03541=1017.922,36.753,-108.696,166.465,54.251,159.872
C03542=1017.928,37.003,-108.711,166.468,54.244,159.872
C03543=1017.934,37.251,-108.726,166.469,54.237,159.871
C03544=1017.939,37.501,-108.741,166.472,54.230,159.870
C03545=1017.944,37.751,-108.756,166.475,54.223,159.869
C03546=1017.949,38.001,-108.771,166.477,54.216,159.868
C03547=1017.955,38.250,-108.786,166.480,54.208,159.867
C03548=1017.961,38.500,-108.801,166.483,54.201,159.867
C03549=1017.966,38.749,-108.816,166.486,54.194,159.866
C03550=1017.971,38.998,-108.832,166.488,54.187,159.865
C03551=1017.977,39.248,-108.846,166.490,54.179,159.864
C03552=1017.982,39.497,-108.862,166.493,54.172,159.863
C03553=1017.987,39.747,-108.876,166.495,54.165,159.862
C03554=1017.993,39.997,-108.892,166.498,54.158,159.862
C03555=1017.998,40.246,-108.906,166.501,54.151,159.861
C03556=1018.003,40.495,-108.921,166.504,54.143,159.860
C03557=1018.009,40.745,-108.937,166.506,54.136,159.859
C03558=1018.014,40.994,-108.952,166.509,54.129,159.858
C03559=1018.020,41.243,-108.967,166.512,54.122,159.858
C03560=1018.026,41.493,-108.982,166.514,54.114,159.857
C03561=1018.031,41.742,-108.997,166.516,54.107,159.856
C03562=1018.036,41.992,-109.013,166.519,54.100,159.855
C03563=1018.042,42.241,-109.028,166.522,54.093,159.854
C03564=1018.047,42.524,-109.045,166.524,54.085,159.853
C03565=1018.053,42.807,-109.063,166.527,54.077,159.852
C03566=1018.059,43.089,-109.080,166.530,54.068,159.851
C03567=1018.066,43.372,-109.097,166.533,54.061,159.851
C03568=1018.071,43.621,-109.113,166.536,54.054,159.850
